  PROC DrawPart23()
    MoveL Offs(pOrigin,281.13,291.37,0.00),v40,z0,tPen\WObj:=wPaper;
    MoveL Offs(pOrigin,281.61,291.85,0.00),v40,z0,tPen\WObj:=wPaper;
    MoveL Offs(pOrigin,281.13,290.89,0.00),v40,z0,tPen\WObj:=wPaper;
    MoveL Offs(pOrigin,281.13,291.37,0.00),v40,z0,tPen\WObj:=wPaper;
    MoveL Offs(pOrigin,281.61,291.85,0.00),v40,fine,tPen\WObj:=wPaper;
    MoveL Offs(pOrigin,281.61,291.85,6.00),v60,z5,tPen\WObj:=wPaper;
    MoveL Offs(pOrigin,262.45,299.03,6.00),vTravel,z5,tPen\WObj:=wPaper;
    MoveL Offs(pOrigin,262.45,299.03,0.00),v60,z0,tPen\WObj:=wPaper;
    MoveL Offs(pOrigin,261.01,295.20,0.00),v40,z0,tPen\WObj:=wPaper;
    MoveL Offs(pOrigin,260.54,294.72,0.00),v40,z0,tPen\WObj:=wPaper;
    MoveL Offs(pOrigin,254.79,294.72,0.00),v40,z0,tPen\WObj:=wPaper;
    MoveL Offs(pOrigin,253.35,295.20,0.00),v40,z0,tPen\WObj:=wPaper;
    MoveL Offs(pOrigin,238.51,295.20,0.00),v40,z0,tPen\WObj:=wPaper;
    MoveL Offs(pOrigin,237.07,294.72,0.00),v40,z0,tPen\WObj:=wPaper;
    MoveL Offs(pOrigin,234.20,294.72,0.00),v40,z0,tPen\WObj:=wPaper;
    MoveL Offs(pOrigin,231.32,293.76,0.00),v40,z0,tPen\WObj:=wPaper;
    MoveL Offs(pOrigin,228.45,293.76,0.00),v40,z0,tPen\WObj:=wPaper;
    MoveL Offs(pOrigin,223.18,292.32,0.00),v40,z0,tPen\WObj:=wPaper;
    MoveL Offs(pOrigin,222.23,292.32,0.00),v40,z0,tPen\WObj:=wPaper;
    MoveL Offs(pOrigin,219.83,291.37,0.00),v40,z0,tPen\WObj:=wPaper;
    MoveL Offs(pOrigin,218.39,291.37,0.00),v40,z0,tPen\WObj:=wPaper;
    MoveL Offs(pOrigin,210.73,288.81,0.00),v40,z0,tPen\WObj:=wPaper;
    MoveL Offs(pOrigin,198.28,282.91,0.00),v40,z0,tPen\WObj:=wPaper;
    MoveL Offs(pOrigin,193.97,280.51,0.00),v40,z0,tPen\WObj:=wPaper;
    MoveL Offs(pOrigin,183.44,273.65,0.00),v40,z0,tPen\WObj:=wPaper;
    MoveL Offs(pOrigin,175.77,267.42,0.00),v40,z0,tPen\WObj:=wPaper;
    MoveL Offs(pOrigin,166.20,257.85,0.00),v40,z0,tPen\WObj:=wPaper;
    MoveL Offs(pOrigin,154.23,242.04,0.00),v40,z0,tPen\WObj:=wPaper;
    MoveL Offs(pOrigin,153.27,241.56,0.00),v40,z0,tPen\WObj:=wPaper;
    MoveL Offs(pOrigin,150.87,242.04,0.00),v40,z0,tPen\WObj:=wPaper;
    MoveL Offs(pOrigin,148.96,241.56,0.00),v40,z0,tPen\WObj:=wPaper;
    MoveL Offs(pOrigin,148.16,242.04,0.00),v40,z0,tPen\WObj:=wPaper;
    MoveL Offs(pOrigin,148.64,243.96,0.00),v40,z0,tPen\WObj:=wPaper;
    MoveL Offs(pOrigin,153.59,253.06,0.00),v40,z0,tPen\WObj:=wPaper;
    MoveL Offs(pOrigin,158.54,260.24,0.00),v40,z0,tPen\WObj:=wPaper;
    MoveL Offs(pOrigin,165.24,268.38,0.00),v40,z0,tPen\WObj:=wPaper;
    MoveL Offs(pOrigin,176.73,279.39,0.00),v40,z0,tPen\WObj:=wPaper;
    MoveL Offs(pOrigin,181.04,282.75,0.00),v40,z0,tPen\WObj:=wPaper;
    MoveL Offs(pOrigin,186.79,286.74,0.00),v40,z0,tPen\WObj:=wPaper;
    MoveL Offs(pOrigin,196.37,292.16,0.00),v40,z0,tPen\WObj:=wPaper;
    MoveL Offs(pOrigin,203.07,295.04,0.00),v40,z0,tPen\WObj:=wPaper;
    MoveL Offs(pOrigin,204.51,296.00,0.00),v40,z0,tPen\WObj:=wPaper;
    MoveL Offs(pOrigin,212.17,298.55,0.00),v40,z0,tPen\WObj:=wPaper;
    MoveL Offs(pOrigin,213.13,298.55,0.00),v40,z0,tPen\WObj:=wPaper;
    MoveL Offs(pOrigin,215.52,299.51,0.00),v40,z0,tPen\WObj:=wPaper;
    MoveL Offs(pOrigin,227.01,302.38,0.00),v40,z0,tPen\WObj:=wPaper;
    MoveL Offs(pOrigin,228.93,302.38,0.00),v40,z0,tPen\WObj:=wPaper;
    MoveL Offs(pOrigin,233.24,303.34,0.00),v40,z0,tPen\WObj:=wPaper;
    MoveL Offs(pOrigin,242.82,303.34,0.00),v40,z0,tPen\WObj:=wPaper;
    MoveL Offs(pOrigin,244.25,303.82,0.00),v40,z0,tPen\WObj:=wPaper;
    MoveL Offs(pOrigin,247.61,303.82,0.00),v40,z0,tPen\WObj:=wPaper;
    MoveL Offs(pOrigin,249.04,303.34,0.00),v40,z0,tPen\WObj:=wPaper;
    MoveL Offs(pOrigin,256.23,303.34,0.00),v40,z0,tPen\WObj:=wPaper;
    MoveL Offs(pOrigin,262.29,301.74,0.00),v40,z0,tPen\WObj:=wPaper;
    MoveL Offs(pOrigin,262.45,299.03,0.00),v40,fine,tPen\WObj:=wPaper;
    MoveL Offs(pOrigin,262.45,299.03,6.00),v60,z5,tPen\WObj:=wPaper;
    MoveL Offs(pOrigin,265.32,312.92,6.00),vTravel,z5,tPen\WObj:=wPaper;
    MoveL Offs(pOrigin,265.32,312.92,0.00),v60,z0,tPen\WObj:=wPaper;
    MoveL Offs(pOrigin,266.28,313.39,0.00),v40,z0,tPen\WObj:=wPaper;
    MoveL Offs(pOrigin,267.08,314.35,0.00),v40,z0,tPen\WObj:=wPaper;
    MoveL Offs(pOrigin,267.40,316.27,0.00),v40,z0,tPen\WObj:=wPaper;
    MoveL Offs(pOrigin,268.68,319.14,0.00),v40,z0,tPen\WObj:=wPaper;
    MoveL Offs(pOrigin,268.20,320.42,0.00),v40,z0,tPen\WObj:=wPaper;
    MoveL Offs(pOrigin,266.76,321.06,0.00),v40,z0,tPen\WObj:=wPaper;
    MoveL Offs(pOrigin,264.85,321.06,0.00),v40,z0,tPen\WObj:=wPaper;
    MoveL Offs(pOrigin,263.41,321.54,0.00),v40,z0,tPen\WObj:=wPaper;
    MoveL Offs(pOrigin,260.06,321.54,0.00),v40,z0,tPen\WObj:=wPaper;
    MoveL Offs(pOrigin,255.75,322.49,0.00),v40,z0,tPen\WObj:=wPaper;
    MoveL Offs(pOrigin,235.63,322.49,0.00),v40,z0,tPen\WObj:=wPaper;
    MoveL Offs(pOrigin,232.28,321.54,0.00),v40,z0,tPen\WObj:=wPaper;
    MoveL Offs(pOrigin,228.45,321.54,0.00),v40,z0,tPen\WObj:=wPaper;
    MoveL Offs(pOrigin,227.01,321.06,0.00),v40,z0,tPen\WObj:=wPaper;
    MoveL Offs(pOrigin,225.10,321.06,0.00),v40,z0,tPen\WObj:=wPaper;
    MoveL Offs(pOrigin,222.23,320.10,0.00),v40,z0,tPen\WObj:=wPaper;
    MoveL Offs(pOrigin,220.31,320.10,0.00),v40,z0,tPen\WObj:=wPaper;
    MoveL Offs(pOrigin,206.90,316.43,0.00),v40,z0,tPen\WObj:=wPaper;
    MoveL Offs(pOrigin,197.32,312.76,0.00),v40,z0,tPen\WObj:=wPaper;
    MoveL Offs(pOrigin,185.83,307.33,0.00),v40,z0,tPen\WObj:=wPaper;
    MoveL Offs(pOrigin,181.04,304.46,0.00),v40,z0,tPen\WObj:=wPaper;
    MoveL Offs(pOrigin,168.59,296.15,0.00),v40,z0,tPen\WObj:=wPaper;
    MoveL Offs(pOrigin,166.20,293.76,0.00),v40,z0,tPen\WObj:=wPaper;
    MoveL Offs(pOrigin,161.41,289.93,0.00),v40,z0,tPen\WObj:=wPaper;
    MoveL Offs(pOrigin,152.31,280.83,0.00),v40,z0,tPen\WObj:=wPaper;
    MoveL Offs(pOrigin,142.25,268.38,0.00),v40,z0,tPen\WObj:=wPaper;
    MoveL Offs(pOrigin,135.71,257.85,0.00),v40,z0,tPen\WObj:=wPaper;
    MoveL Offs(pOrigin,131.88,250.66,0.00),v40,z0,tPen\WObj:=wPaper;
    MoveL Offs(pOrigin,128.69,243.48,0.00),v40,z0,tPen\WObj:=wPaper;
    MoveL Offs(pOrigin,126.29,237.25,0.00),v40,z0,tPen\WObj:=wPaper;
    MoveL Offs(pOrigin,123.58,228.63,0.00),v40,z0,tPen\WObj:=wPaper;
    MoveL Offs(pOrigin,123.58,227.68,0.00),v40,z0,tPen\WObj:=wPaper;
    MoveL Offs(pOrigin,122.62,225.28,0.00),v40,z0,tPen\WObj:=wPaper;
    MoveL Offs(pOrigin,122.14,221.93,0.00),v40,z0,tPen\WObj:=wPaper;
    MoveL Offs(pOrigin,121.18,219.06,0.00),v40,z0,tPen\WObj:=wPaper;
    MoveL Offs(pOrigin,121.18,217.14,0.00),v40,z0,tPen\WObj:=wPaper;
    MoveL Offs(pOrigin,120.23,213.79,0.00),v40,z0,tPen\WObj:=wPaper;
    MoveL Offs(pOrigin,120.23,211.87,0.00),v40,z0,tPen\WObj:=wPaper;
    MoveL Offs(pOrigin,119.75,210.44,0.00),v40,z0,tPen\WObj:=wPaper;
    MoveL Offs(pOrigin,119.75,207.56,0.00),v40,z0,tPen\WObj:=wPaper;
    MoveL Offs(pOrigin,118.79,203.73,0.00),v40,z0,tPen\WObj:=wPaper;
    MoveL Offs(pOrigin,118.79,185.54,0.00),v40,z0,tPen\WObj:=wPaper;
    MoveL Offs(pOrigin,119.27,184.10,0.00),v40,z0,tPen\WObj:=wPaper;
    MoveL Offs(pOrigin,119.27,182.66,0.00),v40,z0,tPen\WObj:=wPaper;
    MoveL Offs(pOrigin,119.75,181.23,0.00),v40,z0,tPen\WObj:=wPaper;
    MoveL Offs(pOrigin,119.75,178.83,0.00),v40,z0,tPen\WObj:=wPaper;
    MoveL Offs(pOrigin,121.18,172.61,0.00),v40,z0,tPen\WObj:=wPaper;
    MoveL Offs(pOrigin,121.18,171.17,0.00),v40,z0,tPen\WObj:=wPaper;
    MoveL Offs(pOrigin,122.62,165.42,0.00),v40,z0,tPen\WObj:=wPaper;
    MoveL Offs(pOrigin,123.10,164.62,0.00),v40,z0,tPen\WObj:=wPaper;
    MoveL Offs(pOrigin,124.06,164.46,0.00),v40,z0,tPen\WObj:=wPaper;
    MoveL Offs(pOrigin,127.89,166.86,0.00),v40,z0,tPen\WObj:=wPaper;
    MoveL Offs(pOrigin,129.32,168.77,0.00),v40,z0,tPen\WObj:=wPaper;
    MoveL Offs(pOrigin,129.32,170.69,0.00),v40,z0,tPen\WObj:=wPaper;
    MoveL Offs(pOrigin,128.37,173.56,0.00),v40,z0,tPen\WObj:=wPaper;
    MoveL Offs(pOrigin,128.37,175.48,0.00),v40,z0,tPen\WObj:=wPaper;
    MoveL Offs(pOrigin,127.41,178.83,0.00),v40,z0,tPen\WObj:=wPaper;
    MoveL Offs(pOrigin,127.41,180.75,0.00),v40,z0,tPen\WObj:=wPaper;
    MoveL Offs(pOrigin,126.93,182.18,0.00),v40,z0,tPen\WObj:=wPaper;
    MoveL Offs(pOrigin,126.93,185.54,0.00),v40,z0,tPen\WObj:=wPaper;
    MoveL Offs(pOrigin,126.45,186.97,0.00),v40,z0,tPen\WObj:=wPaper;
    MoveL Offs(pOrigin,126.45,189.37,0.00),v40,z0,tPen\WObj:=wPaper;
  ENDPROC

  PROC DrawPart24()
    MoveL Offs(pOrigin,125.97,190.80,0.00),v40,z0,tPen\WObj:=wPaper;
    MoveL Offs(pOrigin,125.97,196.55,0.00),v40,z0,tPen\WObj:=wPaper;
    MoveL Offs(pOrigin,126.45,197.99,0.00),v40,z0,tPen\WObj:=wPaper;
    MoveL Offs(pOrigin,126.45,201.82,0.00),v40,z0,tPen\WObj:=wPaper;
    MoveL Offs(pOrigin,126.93,203.25,0.00),v40,z0,tPen\WObj:=wPaper;
    MoveL Offs(pOrigin,126.93,207.56,0.00),v40,z0,tPen\WObj:=wPaper;
    MoveL Offs(pOrigin,127.41,209.00,0.00),v40,z0,tPen\WObj:=wPaper;
    MoveL Offs(pOrigin,127.41,210.92,0.00),v40,z0,tPen\WObj:=wPaper;
    MoveL Offs(pOrigin,128.37,214.27,0.00),v40,z0,tPen\WObj:=wPaper;
    MoveL Offs(pOrigin,128.37,216.66,0.00),v40,z0,tPen\WObj:=wPaper;
    MoveL Offs(pOrigin,132.20,231.51,0.00),v40,z0,tPen\WObj:=wPaper;
    MoveL Offs(pOrigin,133.00,232.94,0.00),v40,z0,tPen\WObj:=wPaper;
    MoveL Offs(pOrigin,133.95,236.30,0.00),v40,z0,tPen\WObj:=wPaper;
    MoveL Offs(pOrigin,137.31,244.44,0.00),v40,z0,tPen\WObj:=wPaper;
    MoveL Offs(pOrigin,141.62,253.06,0.00),v40,z0,tPen\WObj:=wPaper;
    MoveL Offs(pOrigin,146.56,261.20,0.00),v40,z0,tPen\WObj:=wPaper;
    MoveL Offs(pOrigin,153.27,270.30,0.00),v40,z0,tPen\WObj:=wPaper;
    MoveL Offs(pOrigin,158.54,276.52,0.00),v40,z0,tPen\WObj:=wPaper;
    MoveL Offs(pOrigin,168.11,285.62,0.00),v40,z0,tPen\WObj:=wPaper;
    MoveL Offs(pOrigin,175.30,291.37,0.00),v40,z0,tPen\WObj:=wPaper;
    MoveL Offs(pOrigin,180.08,294.72,0.00),v40,z0,tPen\WObj:=wPaper;
    MoveL Offs(pOrigin,190.14,300.78,0.00),v40,z0,tPen\WObj:=wPaper;
    MoveL Offs(pOrigin,196.85,303.98,0.00),v40,z0,tPen\WObj:=wPaper;
    MoveL Offs(pOrigin,201.95,305.89,0.00),v40,z0,tPen\WObj:=wPaper;
    MoveL Offs(pOrigin,204.51,307.33,0.00),v40,z0,tPen\WObj:=wPaper;
    MoveL Offs(pOrigin,207.86,308.29,0.00),v40,z0,tPen\WObj:=wPaper;
    MoveL Offs(pOrigin,209.30,309.08,0.00),v40,z0,tPen\WObj:=wPaper;
    MoveL Offs(pOrigin,210.25,309.08,0.00),v40,z0,tPen\WObj:=wPaper;
    MoveL Offs(pOrigin,214.56,310.52,0.00),v40,z0,tPen\WObj:=wPaper;
    MoveL Offs(pOrigin,216.00,310.52,0.00),v40,z0,tPen\WObj:=wPaper;
    MoveL Offs(pOrigin,218.39,311.48,0.00),v40,z0,tPen\WObj:=wPaper;
    MoveL Offs(pOrigin,221.75,311.96,0.00),v40,z0,tPen\WObj:=wPaper;
    MoveL Offs(pOrigin,225.10,312.92,0.00),v40,z0,tPen\WObj:=wPaper;
    MoveL Offs(pOrigin,227.49,312.92,0.00),v40,z0,tPen\WObj:=wPaper;
    MoveL Offs(pOrigin,231.32,313.87,0.00),v40,z0,tPen\WObj:=wPaper;
    MoveL Offs(pOrigin,234.20,313.87,0.00),v40,z0,tPen\WObj:=wPaper;
    MoveL Offs(pOrigin,235.63,314.35,0.00),v40,z0,tPen\WObj:=wPaper;
    MoveL Offs(pOrigin,242.82,314.35,0.00),v40,z0,tPen\WObj:=wPaper;
    MoveL Offs(pOrigin,244.25,314.83,0.00),v40,z0,tPen\WObj:=wPaper;
    MoveL Offs(pOrigin,248.08,314.83,0.00),v40,z0,tPen\WObj:=wPaper;
    MoveL Offs(pOrigin,249.52,314.35,0.00),v40,z0,tPen\WObj:=wPaper;
    MoveL Offs(pOrigin,256.23,314.35,0.00),v40,z0,tPen\WObj:=wPaper;
    MoveL Offs(pOrigin,257.66,313.87,0.00),v40,z0,tPen\WObj:=wPaper;
    MoveL Offs(pOrigin,260.54,313.87,0.00),v40,z0,tPen\WObj:=wPaper;
    MoveL Offs(pOrigin,265.32,312.92,0.00),v40,fine,tPen\WObj:=wPaper;
    MoveL Offs(pOrigin,265.32,312.92,6.00),v60,z5,tPen\WObj:=wPaper;
    MoveL Offs(pOrigin,280.65,317.70,6.00),vTravel,z5,tPen\WObj:=wPaper;
    MoveL Offs(pOrigin,280.65,317.70,0.00),v60,z0,tPen\WObj:=wPaper;
    MoveL Offs(pOrigin,281.45,319.14,0.00),v40,z0,tPen\WObj:=wPaper;
    MoveL Offs(pOrigin,283.04,325.37,0.00),v40,z0,tPen\WObj:=wPaper;
    MoveL Offs(pOrigin,283.84,326.80,0.00),v40,z0,tPen\WObj:=wPaper;
    MoveL Offs(pOrigin,285.12,330.63,0.00),v40,z0,tPen\WObj:=wPaper;
    MoveL Offs(pOrigin,285.92,331.43,0.00),v40,z0,tPen\WObj:=wPaper;
    MoveL Offs(pOrigin,286.87,331.59,0.00),v40,z0,tPen\WObj:=wPaper;
    MoveL Offs(pOrigin,282.88,322.17,0.00),v40,z0,tPen\WObj:=wPaper;
    MoveL Offs(pOrigin,280.65,317.70,0.00),v40,fine,tPen\WObj:=wPaper;
    MoveL Offs(pOrigin,280.65,317.70,6.00),v60,z5,tPen\WObj:=wPaper;
    MoveL Offs(pOrigin,288.31,331.43,6.00),vTravel,z5,tPen\WObj:=wPaper;
    MoveL Offs(pOrigin,288.31,331.43,0.00),v60,z0,tPen\WObj:=wPaper;
    MoveL Offs(pOrigin,291.66,330.47,0.00),v40,z0,tPen\WObj:=wPaper;
    MoveL Offs(pOrigin,298.37,327.44,0.00),v40,z0,tPen\WObj:=wPaper;
    MoveL Offs(pOrigin,299.80,327.12,0.00),v40,z0,tPen\WObj:=wPaper;
    MoveL Offs(pOrigin,306.83,323.29,0.00),v40,z0,tPen\WObj:=wPaper;
    MoveL Offs(pOrigin,288.31,331.43,0.00),v40,fine,tPen\WObj:=wPaper;
    MoveL Offs(pOrigin,288.31,331.43,6.00),v60,z5,tPen\WObj:=wPaper;
    MoveL Offs(pOrigin,297.41,327.76,6.00),vTravel,z5,tPen\WObj:=wPaper;
    MoveL Offs(pOrigin,297.41,327.76,0.00),v60,z0,tPen\WObj:=wPaper;
    MoveL Offs(pOrigin,297.89,327.28,0.00),v40,z0,tPen\WObj:=wPaper;
    MoveL Offs(pOrigin,297.89,327.76,0.00),v40,z0,tPen\WObj:=wPaper;
    MoveL Offs(pOrigin,297.41,327.76,0.00),v40,z0,tPen\WObj:=wPaper;
    MoveL Offs(pOrigin,297.89,327.28,0.00),v40,z0,tPen\WObj:=wPaper;
    MoveL Offs(pOrigin,297.89,327.76,0.00),v40,z0,tPen\WObj:=wPaper;
    MoveL Offs(pOrigin,297.41,327.76,0.00),v40,fine,tPen\WObj:=wPaper;
    MoveL Offs(pOrigin,297.41,327.76,6.00),v60,z5,tPen\WObj:=wPaper;
    MoveL Offs(pOrigin,302.68,325.37,6.00),vTravel,z5,tPen\WObj:=wPaper;
    MoveL Offs(pOrigin,302.68,325.37,0.00),v60,z0,tPen\WObj:=wPaper;
    MoveL Offs(pOrigin,303.15,324.89,0.00),v40,z0,tPen\WObj:=wPaper;
    MoveL Offs(pOrigin,303.15,325.37,0.00),v40,z0,tPen\WObj:=wPaper;
    MoveL Offs(pOrigin,302.68,325.37,0.00),v40,z0,tPen\WObj:=wPaper;
    MoveL Offs(pOrigin,303.15,324.89,0.00),v40,z0,tPen\WObj:=wPaper;
    MoveL Offs(pOrigin,303.15,325.37,0.00),v40,z0,tPen\WObj:=wPaper;
    MoveL Offs(pOrigin,302.68,325.37,0.00),v40,fine,tPen\WObj:=wPaper;
    MoveL Offs(pOrigin,302.68,325.37,6.00),v60,z5,tPen\WObj:=wPaper;
    MoveL Offs(pOrigin,307.94,322.81,6.00),vTravel,z5,tPen\WObj:=wPaper;
    MoveL Offs(pOrigin,307.94,322.81,0.00),v60,z0,tPen\WObj:=wPaper;
    MoveL Offs(pOrigin,321.35,314.83,0.00),v40,z0,tPen\WObj:=wPaper;
    MoveL Offs(pOrigin,321.99,314.03,0.00),v40,z0,tPen\WObj:=wPaper;
    MoveL Offs(pOrigin,307.94,322.81,0.00),v40,fine,tPen\WObj:=wPaper;
    MoveL Offs(pOrigin,307.94,322.81,6.00),v60,z5,tPen\WObj:=wPaper;
    MoveL Offs(pOrigin,308.90,322.01,6.00),vTravel,z5,tPen\WObj:=wPaper;
    MoveL Offs(pOrigin,308.90,322.01,0.00),v60,z0,tPen\WObj:=wPaper;
    MoveL Offs(pOrigin,309.38,321.54,0.00),v40,z0,tPen\WObj:=wPaper;
    MoveL Offs(pOrigin,309.38,322.01,0.00),v40,z0,tPen\WObj:=wPaper;
    MoveL Offs(pOrigin,308.90,322.01,0.00),v40,z0,tPen\WObj:=wPaper;
    MoveL Offs(pOrigin,309.38,321.54,0.00),v40,z0,tPen\WObj:=wPaper;
    MoveL Offs(pOrigin,309.38,322.01,0.00),v40,z0,tPen\WObj:=wPaper;
    MoveL Offs(pOrigin,308.90,322.01,0.00),v40,fine,tPen\WObj:=wPaper;
    MoveL Offs(pOrigin,308.90,322.01,6.00),v60,z5,tPen\WObj:=wPaper;
    MoveL Offs(pOrigin,313.21,319.62,6.00),vTravel,z5,tPen\WObj:=wPaper;
    MoveL Offs(pOrigin,313.21,319.62,0.00),v60,z0,tPen\WObj:=wPaper;
    MoveL Offs(pOrigin,313.69,319.14,0.00),v40,z0,tPen\WObj:=wPaper;
    MoveL Offs(pOrigin,313.69,319.62,0.00),v40,z0,tPen\WObj:=wPaper;
    MoveL Offs(pOrigin,313.21,319.62,0.00),v40,z0,tPen\WObj:=wPaper;
    MoveL Offs(pOrigin,313.69,319.14,0.00),v40,z0,tPen\WObj:=wPaper;
    MoveL Offs(pOrigin,313.69,319.62,0.00),v40,z0,tPen\WObj:=wPaper;
    MoveL Offs(pOrigin,313.21,319.62,0.00),v40,fine,tPen\WObj:=wPaper;
    MoveL Offs(pOrigin,313.21,319.62,6.00),v60,z5,tPen\WObj:=wPaper;
    MoveL Offs(pOrigin,314.65,318.66,6.00),vTravel,z5,tPen\WObj:=wPaper;
    MoveL Offs(pOrigin,314.65,318.66,0.00),v60,z0,tPen\WObj:=wPaper;
    MoveL Offs(pOrigin,315.13,318.18,0.00),v40,z0,tPen\WObj:=wPaper;
    MoveL Offs(pOrigin,315.13,318.66,0.00),v40,z0,tPen\WObj:=wPaper;
    MoveL Offs(pOrigin,314.65,318.66,0.00),v40,z0,tPen\WObj:=wPaper;
    MoveL Offs(pOrigin,315.13,318.18,0.00),v40,z0,tPen\WObj:=wPaper;
    MoveL Offs(pOrigin,315.13,318.66,0.00),v40,z0,tPen\WObj:=wPaper;
    MoveL Offs(pOrigin,314.65,318.66,0.00),v40,fine,tPen\WObj:=wPaper;
    MoveL Offs(pOrigin,314.65,318.66,6.00),v60,z5,tPen\WObj:=wPaper;
    MoveL Offs(pOrigin,317.04,317.23,6.00),vTravel,z5,tPen\WObj:=wPaper;
    MoveL Offs(pOrigin,317.04,317.23,0.00),v60,z0,tPen\WObj:=wPaper;
    MoveL Offs(pOrigin,317.52,316.75,0.00),v40,z0,tPen\WObj:=wPaper;
    MoveL Offs(pOrigin,317.52,317.23,0.00),v40,z0,tPen\WObj:=wPaper;
  ENDPROC

  PROC DrawPart25()
    MoveL Offs(pOrigin,317.04,317.23,0.00),v40,z0,tPen\WObj:=wPaper;
    MoveL Offs(pOrigin,317.52,316.75,0.00),v40,z0,tPen\WObj:=wPaper;
    MoveL Offs(pOrigin,317.52,317.23,0.00),v40,z0,tPen\WObj:=wPaper;
    MoveL Offs(pOrigin,317.04,317.23,0.00),v40,fine,tPen\WObj:=wPaper;
    MoveL Offs(pOrigin,317.04,317.23,6.00),v60,z5,tPen\WObj:=wPaper;
    MoveL Offs(pOrigin,312.25,310.04,6.00),vTravel,z5,tPen\WObj:=wPaper;
    MoveL Offs(pOrigin,312.25,310.04,0.00),v60,z0,tPen\WObj:=wPaper;
    MoveL Offs(pOrigin,311.77,310.04,0.00),v40,z0,tPen\WObj:=wPaper;
    MoveL Offs(pOrigin,312.25,309.56,0.00),v40,z0,tPen\WObj:=wPaper;
    MoveL Offs(pOrigin,312.25,310.04,0.00),v40,z0,tPen\WObj:=wPaper;
    MoveL Offs(pOrigin,311.77,310.04,0.00),v40,z0,tPen\WObj:=wPaper;
    MoveL Offs(pOrigin,312.25,309.56,0.00),v40,z0,tPen\WObj:=wPaper;
    MoveL Offs(pOrigin,312.25,310.04,0.00),v40,fine,tPen\WObj:=wPaper;
    MoveL Offs(pOrigin,312.25,310.04,6.00),v60,z5,tPen\WObj:=wPaper;
    MoveL Offs(pOrigin,310.82,310.52,6.00),vTravel,z5,tPen\WObj:=wPaper;
    MoveL Offs(pOrigin,310.82,310.52,0.00),v60,z0,tPen\WObj:=wPaper;
    MoveL Offs(pOrigin,310.82,311.00,0.00),v40,z0,tPen\WObj:=wPaper;
    MoveL Offs(pOrigin,310.34,311.00,0.00),v40,z0,tPen\WObj:=wPaper;
    MoveL Offs(pOrigin,310.82,310.52,0.00),v40,z0,tPen\WObj:=wPaper;
    MoveL Offs(pOrigin,310.82,311.00,0.00),v40,z0,tPen\WObj:=wPaper;
    MoveL Offs(pOrigin,310.34,311.00,0.00),v40,z0,tPen\WObj:=wPaper;
    MoveL Offs(pOrigin,310.82,310.52,0.00),v40,fine,tPen\WObj:=wPaper;
    MoveL Offs(pOrigin,310.82,310.52,6.00),v60,z5,tPen\WObj:=wPaper;
    MoveL Offs(pOrigin,317.04,306.69,6.00),vTravel,z5,tPen\WObj:=wPaper;
    MoveL Offs(pOrigin,317.04,306.69,0.00),v60,z0,tPen\WObj:=wPaper;
    MoveL Offs(pOrigin,318.00,305.73,0.00),v40,z0,tPen\WObj:=wPaper;
    MoveL Offs(pOrigin,318.00,306.21,0.00),v40,z0,tPen\WObj:=wPaper;
    MoveL Offs(pOrigin,317.52,306.21,0.00),v40,z0,tPen\WObj:=wPaper;
    MoveL Offs(pOrigin,317.04,306.69,0.00),v40,z0,tPen\WObj:=wPaper;
    MoveL Offs(pOrigin,318.00,305.73,0.00),v40,z0,tPen\WObj:=wPaper;
    MoveL Offs(pOrigin,318.00,306.21,0.00),v40,z0,tPen\WObj:=wPaper;
    MoveL Offs(pOrigin,317.52,306.21,0.00),v40,z0,tPen\WObj:=wPaper;
    MoveL Offs(pOrigin,317.04,306.69,0.00),v40,fine,tPen\WObj:=wPaper;
    MoveL Offs(pOrigin,317.04,306.69,6.00),v60,z5,tPen\WObj:=wPaper;
    MoveL Offs(pOrigin,318.96,305.25,6.00),vTravel,z5,tPen\WObj:=wPaper;
    MoveL Offs(pOrigin,318.96,305.25,0.00),v60,z0,tPen\WObj:=wPaper;
    MoveL Offs(pOrigin,319.44,304.77,0.00),v40,z0,tPen\WObj:=wPaper;
    MoveL Offs(pOrigin,319.44,305.25,0.00),v40,z0,tPen\WObj:=wPaper;
    MoveL Offs(pOrigin,318.96,305.25,0.00),v40,z0,tPen\WObj:=wPaper;
    MoveL Offs(pOrigin,319.44,304.77,0.00),v40,z0,tPen\WObj:=wPaper;
    MoveL Offs(pOrigin,319.44,305.25,0.00),v40,z0,tPen\WObj:=wPaper;
    MoveL Offs(pOrigin,318.96,305.25,0.00),v40,fine,tPen\WObj:=wPaper;
    MoveL Offs(pOrigin,318.96,305.25,6.00),v60,z5,tPen\WObj:=wPaper;
    MoveL Offs(pOrigin,320.39,304.30,6.00),vTravel,z5,tPen\WObj:=wPaper;
    MoveL Offs(pOrigin,320.39,304.30,0.00),v60,z0,tPen\WObj:=wPaper;
    MoveL Offs(pOrigin,321.35,303.34,0.00),v40,z0,tPen\WObj:=wPaper;
    MoveL Offs(pOrigin,321.35,303.82,0.00),v40,z0,tPen\WObj:=wPaper;
    MoveL Offs(pOrigin,320.87,303.82,0.00),v40,z0,tPen\WObj:=wPaper;
    MoveL Offs(pOrigin,320.39,304.30,0.00),v40,z0,tPen\WObj:=wPaper;
    MoveL Offs(pOrigin,321.35,303.34,0.00),v40,z0,tPen\WObj:=wPaper;
    MoveL Offs(pOrigin,321.35,303.82,0.00),v40,z0,tPen\WObj:=wPaper;
    MoveL Offs(pOrigin,320.87,303.82,0.00),v40,z0,tPen\WObj:=wPaper;
    MoveL Offs(pOrigin,320.39,304.30,0.00),v40,fine,tPen\WObj:=wPaper;
    MoveL Offs(pOrigin,320.39,304.30,6.00),v60,z5,tPen\WObj:=wPaper;
    MoveL Offs(pOrigin,322.79,302.38,6.00),vTravel,z5,tPen\WObj:=wPaper;
    MoveL Offs(pOrigin,322.79,302.38,0.00),v60,z0,tPen\WObj:=wPaper;
    MoveL Offs(pOrigin,323.75,301.42,0.00),v40,z0,tPen\WObj:=wPaper;
    MoveL Offs(pOrigin,323.75,301.90,0.00),v40,z0,tPen\WObj:=wPaper;
    MoveL Offs(pOrigin,323.27,301.90,0.00),v40,z0,tPen\WObj:=wPaper;
    MoveL Offs(pOrigin,322.79,302.38,0.00),v40,z0,tPen\WObj:=wPaper;
    MoveL Offs(pOrigin,323.75,301.42,0.00),v40,z0,tPen\WObj:=wPaper;
    MoveL Offs(pOrigin,323.75,301.90,0.00),v40,z0,tPen\WObj:=wPaper;
    MoveL Offs(pOrigin,323.27,301.90,0.00),v40,z0,tPen\WObj:=wPaper;
    MoveL Offs(pOrigin,322.79,302.38,0.00),v40,fine,tPen\WObj:=wPaper;
    MoveL Offs(pOrigin,322.79,302.38,6.00),v60,z5,tPen\WObj:=wPaper;
    MoveL Offs(pOrigin,324.70,300.94,6.00),vTravel,z5,tPen\WObj:=wPaper;
    MoveL Offs(pOrigin,324.70,300.94,0.00),v60,z0,tPen\WObj:=wPaper;
    MoveL Offs(pOrigin,325.66,299.99,0.00),v40,z0,tPen\WObj:=wPaper;
    MoveL Offs(pOrigin,325.66,300.46,0.00),v40,z0,tPen\WObj:=wPaper;
    MoveL Offs(pOrigin,325.18,300.46,0.00),v40,z0,tPen\WObj:=wPaper;
    MoveL Offs(pOrigin,324.70,300.94,0.00),v40,z0,tPen\WObj:=wPaper;
    MoveL Offs(pOrigin,325.66,299.99,0.00),v40,z0,tPen\WObj:=wPaper;
    MoveL Offs(pOrigin,325.66,300.46,0.00),v40,z0,tPen\WObj:=wPaper;
    MoveL Offs(pOrigin,325.18,300.46,0.00),v40,z0,tPen\WObj:=wPaper;
    MoveL Offs(pOrigin,324.70,300.94,0.00),v40,fine,tPen\WObj:=wPaper;
    MoveL Offs(pOrigin,324.70,300.94,6.00),v60,z5,tPen\WObj:=wPaper;
    MoveL Offs(pOrigin,331.89,306.21,6.00),vTravel,z5,tPen\WObj:=wPaper;
    MoveL Offs(pOrigin,331.89,306.21,0.00),v60,z0,tPen\WObj:=wPaper;
    MoveL Offs(pOrigin,331.89,306.69,0.00),v40,z0,tPen\WObj:=wPaper;
    MoveL Offs(pOrigin,331.41,307.17,0.00),v40,z0,tPen\WObj:=wPaper;
    MoveL Offs(pOrigin,331.89,306.21,0.00),v40,z0,tPen\WObj:=wPaper;
    MoveL Offs(pOrigin,331.89,306.69,0.00),v40,z0,tPen\WObj:=wPaper;
    MoveL Offs(pOrigin,331.41,307.17,0.00),v40,z0,tPen\WObj:=wPaper;
    MoveL Offs(pOrigin,331.89,306.21,0.00),v40,z0,tPen\WObj:=wPaper;
    MoveL Offs(pOrigin,332.85,305.73,0.00),v40,z0,tPen\WObj:=wPaper;
    MoveL Offs(pOrigin,333.80,304.77,0.00),v40,z0,tPen\WObj:=wPaper;
    MoveL Offs(pOrigin,332.85,305.73,0.00),v40,fine,tPen\WObj:=wPaper;
    MoveL Offs(pOrigin,332.85,305.73,6.00),v60,z5,tPen\WObj:=wPaper;
    MoveL Offs(pOrigin,334.76,304.30,6.00),vTravel,z5,tPen\WObj:=wPaper;
    MoveL Offs(pOrigin,334.76,304.30,0.00),v60,z0,tPen\WObj:=wPaper;
    MoveL Offs(pOrigin,335.24,303.82,0.00),v40,z0,tPen\WObj:=wPaper;
    MoveL Offs(pOrigin,335.24,303.34,0.00),v40,z0,tPen\WObj:=wPaper;
    MoveL Offs(pOrigin,334.76,304.30,0.00),v40,z0,tPen\WObj:=wPaper;
    MoveL Offs(pOrigin,335.24,303.82,0.00),v40,z0,tPen\WObj:=wPaper;
    MoveL Offs(pOrigin,335.24,303.34,0.00),v40,z0,tPen\WObj:=wPaper;
    MoveL Offs(pOrigin,334.76,304.30,0.00),v40,fine,tPen\WObj:=wPaper;
    MoveL Offs(pOrigin,334.76,304.30,6.00),v60,z5,tPen\WObj:=wPaper;
    MoveL Offs(pOrigin,336.20,302.86,6.00),vTravel,z5,tPen\WObj:=wPaper;
    MoveL Offs(pOrigin,336.20,302.86,0.00),v60,z0,tPen\WObj:=wPaper;
    MoveL Offs(pOrigin,336.68,302.38,0.00),v40,z0,tPen\WObj:=wPaper;
    MoveL Offs(pOrigin,336.68,301.90,0.00),v40,z0,tPen\WObj:=wPaper;
    MoveL Offs(pOrigin,336.20,302.86,0.00),v40,z0,tPen\WObj:=wPaper;
    MoveL Offs(pOrigin,336.68,302.38,0.00),v40,z0,tPen\WObj:=wPaper;
    MoveL Offs(pOrigin,336.68,301.90,0.00),v40,z0,tPen\WObj:=wPaper;
    MoveL Offs(pOrigin,336.20,302.86,0.00),v40,fine,tPen\WObj:=wPaper;
    MoveL Offs(pOrigin,336.20,302.86,6.00),v60,z5,tPen\WObj:=wPaper;
    MoveL Offs(pOrigin,338.59,300.94,6.00),vTravel,z5,tPen\WObj:=wPaper;
    MoveL Offs(pOrigin,338.59,300.94,0.00),v60,z0,tPen\WObj:=wPaper;
    MoveL Offs(pOrigin,339.07,300.46,0.00),v40,z0,tPen\WObj:=wPaper;
    MoveL Offs(pOrigin,339.07,299.99,0.00),v40,z0,tPen\WObj:=wPaper;
    MoveL Offs(pOrigin,338.59,300.94,0.00),v40,z0,tPen\WObj:=wPaper;
    MoveL Offs(pOrigin,339.07,300.46,0.00),v40,z0,tPen\WObj:=wPaper;
    MoveL Offs(pOrigin,339.07,299.99,0.00),v40,z0,tPen\WObj:=wPaper;
    MoveL Offs(pOrigin,338.59,300.94,0.00),v40,fine,tPen\WObj:=wPaper;
    MoveL Offs(pOrigin,338.59,300.94,6.00),v60,z5,tPen\WObj:=wPaper;
    MoveL Offs(pOrigin,340.03,299.51,6.00),vTravel,z5,tPen\WObj:=wPaper;
    MoveL Offs(pOrigin,340.03,299.51,0.00),v60,z0,tPen\WObj:=wPaper;
    MoveL Offs(pOrigin,340.51,299.03,0.00),v40,z0,tPen\WObj:=wPaper;
    MoveL Offs(pOrigin,340.51,298.55,0.00),v40,z0,tPen\WObj:=wPaper;
    MoveL Offs(pOrigin,340.03,299.51,0.00),v40,z0,tPen\WObj:=wPaper;
  ENDPROC

  PROC DrawPart26()
    MoveL Offs(pOrigin,340.51,299.03,0.00),v40,z0,tPen\WObj:=wPaper;
    MoveL Offs(pOrigin,340.51,298.55,0.00),v40,z0,tPen\WObj:=wPaper;
    MoveL Offs(pOrigin,340.03,299.51,0.00),v40,fine,tPen\WObj:=wPaper;
    MoveL Offs(pOrigin,340.03,299.51,6.00),v60,z5,tPen\WObj:=wPaper;
    MoveL Offs(pOrigin,341.46,298.07,6.00),vTravel,z5,tPen\WObj:=wPaper;
    MoveL Offs(pOrigin,341.46,298.07,0.00),v60,z0,tPen\WObj:=wPaper;
    MoveL Offs(pOrigin,341.94,297.59,0.00),v40,z0,tPen\WObj:=wPaper;
    MoveL Offs(pOrigin,341.94,297.11,0.00),v40,z0,tPen\WObj:=wPaper;
    MoveL Offs(pOrigin,341.46,298.07,0.00),v40,z0,tPen\WObj:=wPaper;
    MoveL Offs(pOrigin,341.94,297.59,0.00),v40,z0,tPen\WObj:=wPaper;
    MoveL Offs(pOrigin,341.94,297.11,0.00),v40,z0,tPen\WObj:=wPaper;
    MoveL Offs(pOrigin,341.46,298.07,0.00),v40,fine,tPen\WObj:=wPaper;
    MoveL Offs(pOrigin,341.46,298.07,6.00),v60,z5,tPen\WObj:=wPaper;
    MoveL Offs(pOrigin,342.90,296.63,6.00),vTravel,z5,tPen\WObj:=wPaper;
    MoveL Offs(pOrigin,342.90,296.63,0.00),v60,z0,tPen\WObj:=wPaper;
    MoveL Offs(pOrigin,343.38,296.15,0.00),v40,z0,tPen\WObj:=wPaper;
    MoveL Offs(pOrigin,343.38,295.68,0.00),v40,z0,tPen\WObj:=wPaper;
    MoveL Offs(pOrigin,342.90,296.63,0.00),v40,z0,tPen\WObj:=wPaper;
    MoveL Offs(pOrigin,343.38,296.15,0.00),v40,z0,tPen\WObj:=wPaper;
    MoveL Offs(pOrigin,343.38,295.68,0.00),v40,z0,tPen\WObj:=wPaper;
    MoveL Offs(pOrigin,342.90,296.63,0.00),v40,fine,tPen\WObj:=wPaper;
    MoveL Offs(pOrigin,342.90,296.63,6.00),v60,z5,tPen\WObj:=wPaper;
    MoveL Offs(pOrigin,345.30,293.76,6.00),vTravel,z5,tPen\WObj:=wPaper;
    MoveL Offs(pOrigin,345.30,293.76,0.00),v60,z0,tPen\WObj:=wPaper;
    MoveL Offs(pOrigin,345.77,292.80,0.00),v40,z0,tPen\WObj:=wPaper;
    MoveL Offs(pOrigin,345.77,293.28,0.00),v40,z0,tPen\WObj:=wPaper;
    MoveL Offs(pOrigin,345.30,293.76,0.00),v40,z0,tPen\WObj:=wPaper;
    MoveL Offs(pOrigin,345.77,292.80,0.00),v40,z0,tPen\WObj:=wPaper;
    MoveL Offs(pOrigin,345.77,293.28,0.00),v40,z0,tPen\WObj:=wPaper;
    MoveL Offs(pOrigin,345.30,293.76,0.00),v40,fine,tPen\WObj:=wPaper;
    MoveL Offs(pOrigin,345.30,293.76,6.00),v60,z5,tPen\WObj:=wPaper;
    MoveL Offs(pOrigin,347.69,290.89,6.00),vTravel,z5,tPen\WObj:=wPaper;
    MoveL Offs(pOrigin,347.69,290.89,0.00),v60,z0,tPen\WObj:=wPaper;
    MoveL Offs(pOrigin,348.17,290.41,0.00),v40,z0,tPen\WObj:=wPaper;
    MoveL Offs(pOrigin,348.17,289.93,0.00),v40,z0,tPen\WObj:=wPaper;
    MoveL Offs(pOrigin,347.69,290.89,0.00),v40,z0,tPen\WObj:=wPaper;
    MoveL Offs(pOrigin,348.17,290.41,0.00),v40,z0,tPen\WObj:=wPaper;
    MoveL Offs(pOrigin,348.17,289.93,0.00),v40,z0,tPen\WObj:=wPaper;
    MoveL Offs(pOrigin,347.69,290.89,0.00),v40,fine,tPen\WObj:=wPaper;
    MoveL Offs(pOrigin,347.69,290.89,6.00),v60,z5,tPen\WObj:=wPaper;
    MoveL Offs(pOrigin,349.13,289.45,6.00),vTravel,z5,tPen\WObj:=wPaper;
    MoveL Offs(pOrigin,349.13,289.45,0.00),v60,z0,tPen\WObj:=wPaper;
    MoveL Offs(pOrigin,349.61,288.49,0.00),v40,z0,tPen\WObj:=wPaper;
    MoveL Offs(pOrigin,349.61,288.97,0.00),v40,z0,tPen\WObj:=wPaper;
    MoveL Offs(pOrigin,349.13,289.45,0.00),v40,z0,tPen\WObj:=wPaper;
    MoveL Offs(pOrigin,349.61,288.49,0.00),v40,z0,tPen\WObj:=wPaper;
    MoveL Offs(pOrigin,349.61,288.97,0.00),v40,z0,tPen\WObj:=wPaper;
    MoveL Offs(pOrigin,349.13,289.45,0.00),v40,fine,tPen\WObj:=wPaper;
    MoveL Offs(pOrigin,349.13,289.45,6.00),v60,z5,tPen\WObj:=wPaper;
    MoveL Offs(pOrigin,350.56,287.54,6.00),vTravel,z5,tPen\WObj:=wPaper;
    MoveL Offs(pOrigin,350.56,287.54,0.00),v60,z0,tPen\WObj:=wPaper;
    MoveL Offs(pOrigin,351.04,286.58,0.00),v40,z0,tPen\WObj:=wPaper;
    MoveL Offs(pOrigin,351.04,287.06,0.00),v40,z0,tPen\WObj:=wPaper;
    MoveL Offs(pOrigin,350.56,287.54,0.00),v40,z0,tPen\WObj:=wPaper;
    MoveL Offs(pOrigin,351.04,286.58,0.00),v40,z0,tPen\WObj:=wPaper;
    MoveL Offs(pOrigin,351.04,287.06,0.00),v40,z0,tPen\WObj:=wPaper;
    MoveL Offs(pOrigin,350.56,287.54,0.00),v40,fine,tPen\WObj:=wPaper;
    MoveL Offs(pOrigin,350.56,287.54,6.00),v60,z5,tPen\WObj:=wPaper;
    MoveL Offs(pOrigin,352.00,285.14,6.00),vTravel,z5,tPen\WObj:=wPaper;
    MoveL Offs(pOrigin,352.00,285.14,0.00),v60,z0,tPen\WObj:=wPaper;
    MoveL Offs(pOrigin,352.48,284.18,0.00),v40,z0,tPen\WObj:=wPaper;
    MoveL Offs(pOrigin,352.48,284.66,0.00),v40,z0,tPen\WObj:=wPaper;
    MoveL Offs(pOrigin,352.00,285.14,0.00),v40,z0,tPen\WObj:=wPaper;
    MoveL Offs(pOrigin,352.48,284.18,0.00),v40,z0,tPen\WObj:=wPaper;
    MoveL Offs(pOrigin,352.48,284.66,0.00),v40,z0,tPen\WObj:=wPaper;
    MoveL Offs(pOrigin,352.00,285.14,0.00),v40,fine,tPen\WObj:=wPaper;
    MoveL Offs(pOrigin,352.00,285.14,6.00),v60,z5,tPen\WObj:=wPaper;
    MoveL Offs(pOrigin,353.44,283.70,6.00),vTravel,z5,tPen\WObj:=wPaper;
    MoveL Offs(pOrigin,353.44,283.70,0.00),v60,z0,tPen\WObj:=wPaper;
    MoveL Offs(pOrigin,353.92,282.75,0.00),v40,z0,tPen\WObj:=wPaper;
    MoveL Offs(pOrigin,353.92,283.23,0.00),v40,z0,tPen\WObj:=wPaper;
    MoveL Offs(pOrigin,353.44,283.70,0.00),v40,z0,tPen\WObj:=wPaper;
    MoveL Offs(pOrigin,353.92,282.75,0.00),v40,z0,tPen\WObj:=wPaper;
    MoveL Offs(pOrigin,353.92,283.23,0.00),v40,z0,tPen\WObj:=wPaper;
    MoveL Offs(pOrigin,353.44,283.70,0.00),v40,fine,tPen\WObj:=wPaper;
    MoveL Offs(pOrigin,353.44,283.70,6.00),v60,z5,tPen\WObj:=wPaper;
    MoveL Offs(pOrigin,355.83,280.35,6.00),vTravel,z5,tPen\WObj:=wPaper;
    MoveL Offs(pOrigin,355.83,280.35,0.00),v60,z0,tPen\WObj:=wPaper;
    MoveL Offs(pOrigin,356.31,279.87,0.00),v40,z0,tPen\WObj:=wPaper;
    MoveL Offs(pOrigin,356.31,279.39,0.00),v40,z0,tPen\WObj:=wPaper;
    MoveL Offs(pOrigin,355.83,280.35,0.00),v40,z0,tPen\WObj:=wPaper;
    MoveL Offs(pOrigin,356.31,279.87,0.00),v40,z0,tPen\WObj:=wPaper;
    MoveL Offs(pOrigin,356.31,279.39,0.00),v40,z0,tPen\WObj:=wPaper;
    MoveL Offs(pOrigin,355.83,280.35,0.00),v40,fine,tPen\WObj:=wPaper;
    MoveL Offs(pOrigin,355.83,280.35,6.00),v60,z5,tPen\WObj:=wPaper;
    MoveL Offs(pOrigin,360.14,273.17,6.00),vTravel,z5,tPen\WObj:=wPaper;
    MoveL Offs(pOrigin,360.14,273.17,0.00),v60,z0,tPen\WObj:=wPaper;
    MoveL Offs(pOrigin,360.62,272.21,0.00),v40,z0,tPen\WObj:=wPaper;
    MoveL Offs(pOrigin,360.62,272.69,0.00),v40,z0,tPen\WObj:=wPaper;
    MoveL Offs(pOrigin,360.14,273.17,0.00),v40,z0,tPen\WObj:=wPaper;
    MoveL Offs(pOrigin,360.62,272.21,0.00),v40,z0,tPen\WObj:=wPaper;
    MoveL Offs(pOrigin,360.62,272.69,0.00),v40,z0,tPen\WObj:=wPaper;
    MoveL Offs(pOrigin,360.14,273.17,0.00),v40,fine,tPen\WObj:=wPaper;
    MoveL Offs(pOrigin,360.14,273.17,6.00),v60,z5,tPen\WObj:=wPaper;
    MoveL Offs(pOrigin,349.61,273.17,6.00),vTravel,z5,tPen\WObj:=wPaper;
    MoveL Offs(pOrigin,349.61,273.17,0.00),v60,z0,tPen\WObj:=wPaper;
    MoveL Offs(pOrigin,348.65,274.13,0.00),v40,z0,tPen\WObj:=wPaper;
    MoveL Offs(pOrigin,349.61,272.69,0.00),v40,z0,tPen\WObj:=wPaper;
    MoveL Offs(pOrigin,349.61,273.17,0.00),v40,z0,tPen\WObj:=wPaper;
    MoveL Offs(pOrigin,348.65,274.13,0.00),v40,z0,tPen\WObj:=wPaper;
    MoveL Offs(pOrigin,349.61,272.69,0.00),v40,z0,tPen\WObj:=wPaper;
    MoveL Offs(pOrigin,349.61,273.17,0.00),v40,fine,tPen\WObj:=wPaper;
    MoveL Offs(pOrigin,349.61,273.17,6.00),v60,z5,tPen\WObj:=wPaper;
    MoveL Offs(pOrigin,348.17,275.08,6.00),vTravel,z5,tPen\WObj:=wPaper;
    MoveL Offs(pOrigin,348.17,275.08,0.00),v60,z0,tPen\WObj:=wPaper;
    MoveL Offs(pOrigin,348.17,275.56,0.00),v40,z0,tPen\WObj:=wPaper;
    MoveL Offs(pOrigin,347.69,276.04,0.00),v40,z0,tPen\WObj:=wPaper;
    MoveL Offs(pOrigin,348.17,275.08,0.00),v40,z0,tPen\WObj:=wPaper;
    MoveL Offs(pOrigin,348.17,275.56,0.00),v40,z0,tPen\WObj:=wPaper;
    MoveL Offs(pOrigin,347.69,276.04,0.00),v40,z0,tPen\WObj:=wPaper;
    MoveL Offs(pOrigin,348.17,275.08,0.00),v40,fine,tPen\WObj:=wPaper;
    MoveL Offs(pOrigin,348.17,275.08,6.00),v60,z5,tPen\WObj:=wPaper;
    MoveL Offs(pOrigin,347.21,276.52,6.00),vTravel,z5,tPen\WObj:=wPaper;
    MoveL Offs(pOrigin,347.21,276.52,0.00),v60,z0,tPen\WObj:=wPaper;
    MoveL Offs(pOrigin,347.21,277.00,0.00),v40,z0,tPen\WObj:=wPaper;
    MoveL Offs(pOrigin,346.25,277.96,0.00),v40,z0,tPen\WObj:=wPaper;
    MoveL Offs(pOrigin,347.21,276.52,0.00),v40,z0,tPen\WObj:=wPaper;
    MoveL Offs(pOrigin,347.21,277.00,0.00),v40,z0,tPen\WObj:=wPaper;
    MoveL Offs(pOrigin,346.25,277.96,0.00),v40,z0,tPen\WObj:=wPaper;
    MoveL Offs(pOrigin,347.21,276.52,0.00),v40,fine,tPen\WObj:=wPaper;
  ENDPROC

  PROC DrawPart27()
    MoveL Offs(pOrigin,347.21,276.52,6.00),v60,z5,tPen\WObj:=wPaper;
    MoveL Offs(pOrigin,344.34,280.83,6.00),vTravel,z5,tPen\WObj:=wPaper;
    MoveL Offs(pOrigin,344.34,280.83,0.00),v60,z0,tPen\WObj:=wPaper;
    MoveL Offs(pOrigin,344.34,281.31,0.00),v40,z0,tPen\WObj:=wPaper;
    MoveL Offs(pOrigin,343.86,281.31,0.00),v40,z0,tPen\WObj:=wPaper;
    MoveL Offs(pOrigin,342.90,282.27,0.00),v40,z0,tPen\WObj:=wPaper;
    MoveL Offs(pOrigin,344.34,280.83,0.00),v40,z0,tPen\WObj:=wPaper;
    MoveL Offs(pOrigin,344.34,281.31,0.00),v40,z0,tPen\WObj:=wPaper;
    MoveL Offs(pOrigin,343.86,281.31,0.00),v40,z0,tPen\WObj:=wPaper;
    MoveL Offs(pOrigin,342.90,282.27,0.00),v40,z0,tPen\WObj:=wPaper;
    MoveL Offs(pOrigin,344.34,280.83,0.00),v40,fine,tPen\WObj:=wPaper;
    MoveL Offs(pOrigin,344.34,280.83,6.00),v60,z5,tPen\WObj:=wPaper;
    MoveL Offs(pOrigin,341.46,284.18,6.00),vTravel,z5,tPen\WObj:=wPaper;
    MoveL Offs(pOrigin,341.46,284.18,0.00),v60,z0,tPen\WObj:=wPaper;
    MoveL Offs(pOrigin,341.46,284.66,0.00),v40,z0,tPen\WObj:=wPaper;
    MoveL Offs(pOrigin,340.99,284.66,0.00),v40,z0,tPen\WObj:=wPaper;
    MoveL Offs(pOrigin,341.46,284.18,0.00),v40,z0,tPen\WObj:=wPaper;
    MoveL Offs(pOrigin,341.46,284.66,0.00),v40,z0,tPen\WObj:=wPaper;
    MoveL Offs(pOrigin,340.99,284.66,0.00),v40,z0,tPen\WObj:=wPaper;
    MoveL Offs(pOrigin,341.46,284.18,0.00),v40,fine,tPen\WObj:=wPaper;
    MoveL Offs(pOrigin,341.46,284.18,6.00),v60,z5,tPen\WObj:=wPaper;
    MoveL Offs(pOrigin,340.51,285.14,6.00),vTravel,z5,tPen\WObj:=wPaper;
    MoveL Offs(pOrigin,340.51,285.14,0.00),v60,z0,tPen\WObj:=wPaper;
    MoveL Offs(pOrigin,340.51,285.62,0.00),v40,z0,tPen\WObj:=wPaper;
    MoveL Offs(pOrigin,340.03,285.62,0.00),v40,z0,tPen\WObj:=wPaper;
    MoveL Offs(pOrigin,340.51,285.14,0.00),v40,z0,tPen\WObj:=wPaper;
    MoveL Offs(pOrigin,340.51,285.62,0.00),v40,z0,tPen\WObj:=wPaper;
    MoveL Offs(pOrigin,340.03,285.62,0.00),v40,z0,tPen\WObj:=wPaper;
    MoveL Offs(pOrigin,340.51,285.14,0.00),v40,fine,tPen\WObj:=wPaper;
    MoveL Offs(pOrigin,340.51,285.14,6.00),v60,z5,tPen\WObj:=wPaper;
    MoveL Offs(pOrigin,338.11,288.01,6.00),vTravel,z5,tPen\WObj:=wPaper;
    MoveL Offs(pOrigin,338.11,288.01,0.00),v60,z0,tPen\WObj:=wPaper;
    MoveL Offs(pOrigin,338.11,288.49,0.00),v40,z0,tPen\WObj:=wPaper;
    MoveL Offs(pOrigin,337.63,288.49,0.00),v40,z0,tPen\WObj:=wPaper;
    MoveL Offs(pOrigin,337.15,288.97,0.00),v40,z0,tPen\WObj:=wPaper;
    MoveL Offs(pOrigin,338.11,288.01,0.00),v40,z0,tPen\WObj:=wPaper;
    MoveL Offs(pOrigin,338.11,288.49,0.00),v40,z0,tPen\WObj:=wPaper;
    MoveL Offs(pOrigin,337.63,288.49,0.00),v40,z0,tPen\WObj:=wPaper;
    MoveL Offs(pOrigin,337.15,288.97,0.00),v40,z0,tPen\WObj:=wPaper;
    MoveL Offs(pOrigin,338.11,288.01,0.00),v40,fine,tPen\WObj:=wPaper;
    MoveL Offs(pOrigin,338.11,288.01,6.00),v60,z5,tPen\WObj:=wPaper;
    MoveL Offs(pOrigin,336.68,289.45,6.00),vTravel,z5,tPen\WObj:=wPaper;
    MoveL Offs(pOrigin,336.68,289.45,0.00),v60,z0,tPen\WObj:=wPaper;
    MoveL Offs(pOrigin,336.68,289.93,0.00),v40,z0,tPen\WObj:=wPaper;
    MoveL Offs(pOrigin,336.20,289.93,0.00),v40,z0,tPen\WObj:=wPaper;
    MoveL Offs(pOrigin,334.28,291.85,0.00),v40,z0,tPen\WObj:=wPaper;
    MoveL Offs(pOrigin,336.68,289.45,0.00),v40,z0,tPen\WObj:=wPaper;
    MoveL Offs(pOrigin,336.68,289.93,0.00),v40,z0,tPen\WObj:=wPaper;
    MoveL Offs(pOrigin,336.20,289.93,0.00),v40,z0,tPen\WObj:=wPaper;
    MoveL Offs(pOrigin,334.28,291.85,0.00),v40,z0,tPen\WObj:=wPaper;
    MoveL Offs(pOrigin,336.68,289.45,0.00),v40,fine,tPen\WObj:=wPaper;
    MoveL Offs(pOrigin,336.68,289.45,6.00),v60,z5,tPen\WObj:=wPaper;
    MoveL Offs(pOrigin,333.80,292.32,6.00),vTravel,z5,tPen\WObj:=wPaper;
    MoveL Offs(pOrigin,333.80,292.32,0.00),v60,z0,tPen\WObj:=wPaper;
    MoveL Offs(pOrigin,333.80,292.80,0.00),v40,z0,tPen\WObj:=wPaper;
    MoveL Offs(pOrigin,333.32,292.80,0.00),v40,z0,tPen\WObj:=wPaper;
    MoveL Offs(pOrigin,332.85,293.28,0.00),v40,z0,tPen\WObj:=wPaper;
    MoveL Offs(pOrigin,333.80,292.32,0.00),v40,z0,tPen\WObj:=wPaper;
    MoveL Offs(pOrigin,333.80,292.80,0.00),v40,z0,tPen\WObj:=wPaper;
    MoveL Offs(pOrigin,333.32,292.80,0.00),v40,z0,tPen\WObj:=wPaper;
    MoveL Offs(pOrigin,332.85,293.28,0.00),v40,z0,tPen\WObj:=wPaper;
    MoveL Offs(pOrigin,333.80,292.32,0.00),v40,fine,tPen\WObj:=wPaper;
    MoveL Offs(pOrigin,333.80,292.32,6.00),v60,z5,tPen\WObj:=wPaper;
    MoveL Offs(pOrigin,332.21,294.08,6.00),vTravel,z5,tPen\WObj:=wPaper;
    MoveL Offs(pOrigin,332.21,294.08,0.00),v60,z0,tPen\WObj:=wPaper;
    MoveL Offs(pOrigin,327.58,298.55,0.00),v40,z0,tPen\WObj:=wPaper;
    MoveL Offs(pOrigin,332.21,294.08,0.00),v40,fine,tPen\WObj:=wPaper;
    MoveL Offs(pOrigin,332.21,294.08,6.00),v60,z5,tPen\WObj:=wPaper;
    MoveL Offs(pOrigin,328.22,283.86,6.00),vTravel,z5,tPen\WObj:=wPaper;
    MoveL Offs(pOrigin,328.22,283.86,0.00),v60,z0,tPen\WObj:=wPaper;
    MoveL Offs(pOrigin,334.28,275.08,0.00),v40,z0,tPen\WObj:=wPaper;
    MoveL Offs(pOrigin,334.12,277.00,0.00),v40,z0,tPen\WObj:=wPaper;
    MoveL Offs(pOrigin,332.69,279.87,0.00),v40,z0,tPen\WObj:=wPaper;
    MoveL Offs(pOrigin,329.49,283.07,0.00),v40,z0,tPen\WObj:=wPaper;
    MoveL Offs(pOrigin,328.54,283.38,0.00),v40,z0,tPen\WObj:=wPaper;
    MoveL Offs(pOrigin,328.22,283.86,0.00),v40,fine,tPen\WObj:=wPaper;
    MoveL Offs(pOrigin,328.22,283.86,6.00),v60,z5,tPen\WObj:=wPaper;
    MoveL Offs(pOrigin,330.45,282.27,6.00),vTravel,z5,tPen\WObj:=wPaper;
    MoveL Offs(pOrigin,330.45,282.27,0.00),v60,z0,tPen\WObj:=wPaper;
    MoveL Offs(pOrigin,330.93,281.79,0.00),v40,z0,tPen\WObj:=wPaper;
    MoveL Offs(pOrigin,330.93,281.31,0.00),v40,z0,tPen\WObj:=wPaper;
    MoveL Offs(pOrigin,330.45,282.27,0.00),v40,z0,tPen\WObj:=wPaper;
    MoveL Offs(pOrigin,330.93,281.79,0.00),v40,z0,tPen\WObj:=wPaper;
    MoveL Offs(pOrigin,330.93,281.31,0.00),v40,z0,tPen\WObj:=wPaper;
    MoveL Offs(pOrigin,330.45,282.27,0.00),v40,fine,tPen\WObj:=wPaper;
    MoveL Offs(pOrigin,330.45,282.27,6.00),v60,z5,tPen\WObj:=wPaper;
    MoveL Offs(pOrigin,331.89,280.83,6.00),vTravel,z5,tPen\WObj:=wPaper;
    MoveL Offs(pOrigin,331.89,280.83,0.00),v60,z0,tPen\WObj:=wPaper;
    MoveL Offs(pOrigin,332.37,280.35,0.00),v40,z0,tPen\WObj:=wPaper;
    MoveL Offs(pOrigin,332.37,279.87,0.00),v40,z0,tPen\WObj:=wPaper;
    MoveL Offs(pOrigin,331.89,280.83,0.00),v40,z0,tPen\WObj:=wPaper;
    MoveL Offs(pOrigin,332.37,280.35,0.00),v40,z0,tPen\WObj:=wPaper;
    MoveL Offs(pOrigin,332.37,279.87,0.00),v40,z0,tPen\WObj:=wPaper;
    MoveL Offs(pOrigin,331.89,280.83,0.00),v40,fine,tPen\WObj:=wPaper;
    MoveL Offs(pOrigin,331.89,280.83,6.00),v60,z5,tPen\WObj:=wPaper;
    MoveL Offs(pOrigin,334.28,273.65,6.00),vTravel,z5,tPen\WObj:=wPaper;
    MoveL Offs(pOrigin,334.28,273.65,0.00),v60,z0,tPen\WObj:=wPaper;
    MoveL Offs(pOrigin,330.93,265.51,0.00),v40,z0,tPen\WObj:=wPaper;
    MoveL Offs(pOrigin,333.00,268.38,0.00),v40,z0,tPen\WObj:=wPaper;
    MoveL Offs(pOrigin,334.12,270.77,0.00),v40,z0,tPen\WObj:=wPaper;
    MoveL Offs(pOrigin,334.28,273.65,0.00),v40,fine,tPen\WObj:=wPaper;
    MoveL Offs(pOrigin,334.28,273.65,6.00),v60,z5,tPen\WObj:=wPaper;
    MoveL Offs(pOrigin,328.06,263.11,6.00),vTravel,z5,tPen\WObj:=wPaper;
    MoveL Offs(pOrigin,328.06,263.11,0.00),v60,z0,tPen\WObj:=wPaper;
    MoveL Offs(pOrigin,327.58,262.63,0.00),v40,z0,tPen\WObj:=wPaper;
    MoveL Offs(pOrigin,327.58,263.11,0.00),v40,z0,tPen\WObj:=wPaper;
    MoveL Offs(pOrigin,328.06,263.11,0.00),v40,z0,tPen\WObj:=wPaper;
    MoveL Offs(pOrigin,327.58,262.63,0.00),v40,z0,tPen\WObj:=wPaper;
    MoveL Offs(pOrigin,327.58,263.11,0.00),v40,z0,tPen\WObj:=wPaper;
    MoveL Offs(pOrigin,328.06,263.11,0.00),v40,fine,tPen\WObj:=wPaper;
    MoveL Offs(pOrigin,328.06,263.11,6.00),v60,z5,tPen\WObj:=wPaper;
    MoveL Offs(pOrigin,340.51,263.11,6.00),vTravel,z5,tPen\WObj:=wPaper;
    MoveL Offs(pOrigin,340.51,263.11,0.00),v60,z0,tPen\WObj:=wPaper;
    MoveL Offs(pOrigin,340.99,263.11,0.00),v40,z0,tPen\WObj:=wPaper;
    MoveL Offs(pOrigin,341.46,263.59,0.00),v40,z0,tPen\WObj:=wPaper;
    MoveL Offs(pOrigin,340.51,263.11,0.00),v40,z0,tPen\WObj:=wPaper;
    MoveL Offs(pOrigin,340.99,263.11,0.00),v40,z0,tPen\WObj:=wPaper;
    MoveL Offs(pOrigin,341.46,263.59,0.00),v40,z0,tPen\WObj:=wPaper;
    MoveL Offs(pOrigin,340.51,263.11,0.00),v40,fine,tPen\WObj:=wPaper;
    MoveL Offs(pOrigin,340.51,263.11,6.00),v60,z5,tPen\WObj:=wPaper;
  ENDPROC

  PROC DrawPart28()
    MoveL Offs(pOrigin,344.34,255.93,6.00),vTravel,z5,tPen\WObj:=wPaper;
    MoveL Offs(pOrigin,344.34,255.93,0.00),v60,z0,tPen\WObj:=wPaper;
    MoveL Offs(pOrigin,344.82,255.93,0.00),v40,z0,tPen\WObj:=wPaper;
    MoveL Offs(pOrigin,344.34,255.45,0.00),v40,z0,tPen\WObj:=wPaper;
    MoveL Offs(pOrigin,344.34,255.93,0.00),v40,z0,tPen\WObj:=wPaper;
    MoveL Offs(pOrigin,344.82,255.93,0.00),v40,z0,tPen\WObj:=wPaper;
    MoveL Offs(pOrigin,344.34,255.45,0.00),v40,z0,tPen\WObj:=wPaper;
    MoveL Offs(pOrigin,344.34,255.93,0.00),v40,fine,tPen\WObj:=wPaper;
    MoveL Offs(pOrigin,344.34,255.93,6.00),v60,z5,tPen\WObj:=wPaper;
    MoveL Offs(pOrigin,355.83,245.87,6.00),vTravel,z5,tPen\WObj:=wPaper;
    MoveL Offs(pOrigin,355.83,245.87,0.00),v60,z0,tPen\WObj:=wPaper;
    MoveL Offs(pOrigin,356.79,246.83,0.00),v40,z0,tPen\WObj:=wPaper;
    MoveL Offs(pOrigin,355.83,245.87,0.00),v40,z0,tPen\WObj:=wPaper;
    MoveL Offs(pOrigin,356.31,245.87,0.00),v40,z0,tPen\WObj:=wPaper;
    MoveL Offs(pOrigin,355.83,244.92,0.00),v40,z0,tPen\WObj:=wPaper;
    MoveL Offs(pOrigin,359.98,235.34,0.00),v40,z0,tPen\WObj:=wPaper;
    MoveL Offs(pOrigin,362.06,229.11,0.00),v40,z0,tPen\WObj:=wPaper;
    MoveL Offs(pOrigin,365.41,216.18,0.00),v40,z0,tPen\WObj:=wPaper;
    MoveL Offs(pOrigin,365.41,213.79,0.00),v40,z0,tPen\WObj:=wPaper;
    MoveL Offs(pOrigin,366.37,209.96,0.00),v40,z0,tPen\WObj:=wPaper;
    MoveL Offs(pOrigin,366.37,206.13,0.00),v40,z0,tPen\WObj:=wPaper;
    MoveL Offs(pOrigin,367.00,203.73,0.00),v40,z0,tPen\WObj:=wPaper;
    MoveL Offs(pOrigin,368.28,202.77,0.00),v40,z0,tPen\WObj:=wPaper;
    MoveL Offs(pOrigin,372.59,203.89,0.00),v40,z0,tPen\WObj:=wPaper;
    MoveL Offs(pOrigin,373.55,205.17,0.00),v40,z0,tPen\WObj:=wPaper;
    MoveL Offs(pOrigin,373.55,209.48,0.00),v40,z0,tPen\WObj:=wPaper;
    MoveL Offs(pOrigin,372.59,213.79,0.00),v40,z0,tPen\WObj:=wPaper;
    MoveL Offs(pOrigin,372.59,217.14,0.00),v40,z0,tPen\WObj:=wPaper;
    MoveL Offs(pOrigin,369.72,229.59,0.00),v40,z0,tPen\WObj:=wPaper;
    MoveL Offs(pOrigin,366.05,240.61,0.00),v40,z0,tPen\WObj:=wPaper;
    MoveL Offs(pOrigin,362.85,247.79,0.00),v40,z0,tPen\WObj:=wPaper;
    MoveL Offs(pOrigin,362.06,248.27,0.00),v40,z0,tPen\WObj:=wPaper;
    MoveL Offs(pOrigin,361.10,248.27,0.00),v40,z0,tPen\WObj:=wPaper;
    MoveL Offs(pOrigin,357.75,246.99,0.00),v40,z0,tPen\WObj:=wPaper;
    MoveL Offs(pOrigin,356.31,245.87,0.00),v40,fine,tPen\WObj:=wPaper;
    MoveL Offs(pOrigin,356.31,245.87,6.00),v60,z5,tPen\WObj:=wPaper;
    MoveL Offs(pOrigin,355.83,243.96,6.00),vTravel,z5,tPen\WObj:=wPaper;
    MoveL Offs(pOrigin,355.83,243.96,0.00),v60,z0,tPen\WObj:=wPaper;
    MoveL Offs(pOrigin,356.31,243.00,0.00),v40,z0,tPen\WObj:=wPaper;
    MoveL Offs(pOrigin,356.31,243.48,0.00),v40,z0,tPen\WObj:=wPaper;
    MoveL Offs(pOrigin,355.83,243.96,0.00),v40,z0,tPen\WObj:=wPaper;
    MoveL Offs(pOrigin,356.31,243.00,0.00),v40,z0,tPen\WObj:=wPaper;
    MoveL Offs(pOrigin,356.31,243.48,0.00),v40,z0,tPen\WObj:=wPaper;
    MoveL Offs(pOrigin,355.83,243.96,0.00),v40,fine,tPen\WObj:=wPaper;
    MoveL Offs(pOrigin,355.83,243.96,6.00),v60,z5,tPen\WObj:=wPaper;
    MoveL Offs(pOrigin,345.77,221.61,6.00),vTravel,z5,tPen\WObj:=wPaper;
    MoveL Offs(pOrigin,345.77,221.61,0.00),v60,z0,tPen\WObj:=wPaper;
    MoveL Offs(pOrigin,347.69,220.49,0.00),v40,z0,tPen\WObj:=wPaper;
    MoveL Offs(pOrigin,349.29,218.58,0.00),v40,z0,tPen\WObj:=wPaper;
    MoveL Offs(pOrigin,350.08,214.75,0.00),v40,z0,tPen\WObj:=wPaper;
    MoveL Offs(pOrigin,349.13,212.35,0.00),v40,z0,tPen\WObj:=wPaper;
    MoveL Offs(pOrigin,346.25,209.48,0.00),v40,z0,tPen\WObj:=wPaper;
    MoveL Offs(pOrigin,342.74,204.69,0.00),v40,z0,tPen\WObj:=wPaper;
    MoveL Offs(pOrigin,341.46,201.34,0.00),v40,z0,tPen\WObj:=wPaper;
    MoveL Offs(pOrigin,341.46,198.94,0.00),v40,z0,tPen\WObj:=wPaper;
    MoveL Offs(pOrigin,341.78,197.99,0.00),v40,z0,tPen\WObj:=wPaper;
    MoveL Offs(pOrigin,344.34,193.68,0.00),v40,z0,tPen\WObj:=wPaper;
    MoveL Offs(pOrigin,351.68,184.10,0.00),v40,z0,tPen\WObj:=wPaper;
    MoveL Offs(pOrigin,352.48,183.62,0.00),v40,z0,tPen\WObj:=wPaper;
    MoveL Offs(pOrigin,353.92,183.62,0.00),v40,z0,tPen\WObj:=wPaper;
    MoveL Offs(pOrigin,358.23,185.22,0.00),v40,z0,tPen\WObj:=wPaper;
    MoveL Offs(pOrigin,362.06,187.45,0.00),v40,z0,tPen\WObj:=wPaper;
    MoveL Offs(pOrigin,364.93,190.32,0.00),v40,z0,tPen\WObj:=wPaper;
    MoveL Offs(pOrigin,367.32,191.76,0.00),v40,z0,tPen\WObj:=wPaper;
    MoveL Offs(pOrigin,370.68,191.76,0.00),v40,z0,tPen\WObj:=wPaper;
    MoveL Offs(pOrigin,372.59,190.80,0.00),v40,z0,tPen\WObj:=wPaper;
    MoveL Offs(pOrigin,374.03,187.45,0.00),v40,z0,tPen\WObj:=wPaper;
    MoveL Offs(pOrigin,374.03,186.01,0.00),v40,z0,tPen\WObj:=wPaper;
    MoveL Offs(pOrigin,373.39,184.10,0.00),v40,z0,tPen\WObj:=wPaper;
    MoveL Offs(pOrigin,370.68,179.79,0.00),v40,z0,tPen\WObj:=wPaper;
    MoveL Offs(pOrigin,369.72,178.83,0.00),v40,z0,tPen\WObj:=wPaper;
    MoveL Offs(pOrigin,364.45,175.32,0.00),v40,z0,tPen\WObj:=wPaper;
    MoveL Offs(pOrigin,357.27,172.45,0.00),v40,z0,tPen\WObj:=wPaper;
    MoveL Offs(pOrigin,356.31,171.65,0.00),v40,z0,tPen\WObj:=wPaper;
    MoveL Offs(pOrigin,355.83,170.69,0.00),v40,z0,tPen\WObj:=wPaper;
    MoveL Offs(pOrigin,355.83,167.82,0.00),v40,z0,tPen\WObj:=wPaper;
    MoveL Offs(pOrigin,354.39,161.59,0.00),v40,z0,tPen\WObj:=wPaper;
    MoveL Offs(pOrigin,351.84,155.85,0.00),v40,z0,tPen\WObj:=wPaper;
    MoveL Offs(pOrigin,349.61,152.49,0.00),v40,z0,tPen\WObj:=wPaper;
    MoveL Offs(pOrigin,343.38,146.27,0.00),v40,z0,tPen\WObj:=wPaper;
    MoveL Offs(pOrigin,339.55,143.71,0.00),v40,z0,tPen\WObj:=wPaper;
    MoveL Offs(pOrigin,332.37,140.52,0.00),v40,z0,tPen\WObj:=wPaper;
    MoveL Offs(pOrigin,331.41,140.52,0.00),v40,z0,tPen\WObj:=wPaper;
    MoveL Offs(pOrigin,326.14,139.08,0.00),v40,z0,tPen\WObj:=wPaper;
    MoveL Offs(pOrigin,323.27,139.08,0.00),v40,z0,tPen\WObj:=wPaper;
    MoveL Offs(pOrigin,321.83,138.61,0.00),v40,z0,tPen\WObj:=wPaper;
    MoveL Offs(pOrigin,317.52,138.61,0.00),v40,z0,tPen\WObj:=wPaper;
    MoveL Offs(pOrigin,316.08,139.08,0.00),v40,z0,tPen\WObj:=wPaper;
    MoveL Offs(pOrigin,313.21,139.08,0.00),v40,z0,tPen\WObj:=wPaper;
    MoveL Offs(pOrigin,306.51,141.32,0.00),v40,z0,tPen\WObj:=wPaper;
    MoveL Offs(pOrigin,305.71,142.12,0.00),v40,z0,tPen\WObj:=wPaper;
    MoveL Offs(pOrigin,333.32,220.97,0.00),v40,z0,tPen\WObj:=wPaper;
    MoveL Offs(pOrigin,335.72,221.93,0.00),v40,z0,tPen\WObj:=wPaper;
    MoveL Offs(pOrigin,338.11,222.41,0.00),v40,z0,tPen\WObj:=wPaper;
    MoveL Offs(pOrigin,342.90,222.41,0.00),v40,z0,tPen\WObj:=wPaper;
    MoveL Offs(pOrigin,345.77,221.61,0.00),v40,fine,tPen\WObj:=wPaper;
    MoveL Offs(pOrigin,345.77,221.61,6.00),v60,z5,tPen\WObj:=wPaper;
    MoveL Offs(pOrigin,347.21,220.49,6.00),vTravel,z5,tPen\WObj:=wPaper;
    MoveL Offs(pOrigin,347.21,220.49,0.00),v60,z0,tPen\WObj:=wPaper;
    MoveL Offs(pOrigin,347.69,220.01,0.00),v40,z0,tPen\WObj:=wPaper;
    MoveL Offs(pOrigin,347.69,220.49,0.00),v40,z0,tPen\WObj:=wPaper;
    MoveL Offs(pOrigin,347.21,220.49,0.00),v40,z0,tPen\WObj:=wPaper;
    MoveL Offs(pOrigin,347.69,220.01,0.00),v40,z0,tPen\WObj:=wPaper;
    MoveL Offs(pOrigin,347.69,220.49,0.00),v40,z0,tPen\WObj:=wPaper;
    MoveL Offs(pOrigin,347.21,220.49,0.00),v40,fine,tPen\WObj:=wPaper;
    MoveL Offs(pOrigin,347.21,220.49,6.00),v60,z5,tPen\WObj:=wPaper;
    MoveL Offs(pOrigin,348.17,219.54,6.00),vTravel,z5,tPen\WObj:=wPaper;
    MoveL Offs(pOrigin,348.17,219.54,0.00),v60,z0,tPen\WObj:=wPaper;
    MoveL Offs(pOrigin,349.13,218.10,0.00),v40,z0,tPen\WObj:=wPaper;
    MoveL Offs(pOrigin,349.13,218.58,0.00),v40,z0,tPen\WObj:=wPaper;
    MoveL Offs(pOrigin,348.17,219.54,0.00),v40,z0,tPen\WObj:=wPaper;
    MoveL Offs(pOrigin,349.13,218.10,0.00),v40,z0,tPen\WObj:=wPaper;
    MoveL Offs(pOrigin,349.13,218.58,0.00),v40,z0,tPen\WObj:=wPaper;
    MoveL Offs(pOrigin,348.17,219.54,0.00),v40,fine,tPen\WObj:=wPaper;
    MoveL Offs(pOrigin,348.17,219.54,6.00),v60,z5,tPen\WObj:=wPaper;
    MoveL Offs(pOrigin,346.25,209.96,6.00),vTravel,z5,tPen\WObj:=wPaper;
    MoveL Offs(pOrigin,346.25,209.96,0.00),v60,z0,tPen\WObj:=wPaper;
    MoveL Offs(pOrigin,349.13,212.83,0.00),v40,z0,tPen\WObj:=wPaper;
    MoveL Offs(pOrigin,346.25,209.96,0.00),v40,fine,tPen\WObj:=wPaper;
    MoveL Offs(pOrigin,346.25,209.96,6.00),v60,z5,tPen\WObj:=wPaper;
  ENDPROC

  PROC DrawPart29()
    MoveL Offs(pOrigin,344.34,207.56,6.00),vTravel,z5,tPen\WObj:=wPaper;
    MoveL Offs(pOrigin,344.34,207.56,0.00),v60,z0,tPen\WObj:=wPaper;
    MoveL Offs(pOrigin,345.30,208.52,0.00),v40,z0,tPen\WObj:=wPaper;
    MoveL Offs(pOrigin,344.34,207.56,0.00),v40,fine,tPen\WObj:=wPaper;
    MoveL Offs(pOrigin,344.34,207.56,6.00),v60,z5,tPen\WObj:=wPaper;
    MoveL Offs(pOrigin,344.34,193.68,6.00),vTravel,z5,tPen\WObj:=wPaper;
    MoveL Offs(pOrigin,344.34,193.68,0.00),v60,z0,tPen\WObj:=wPaper;
    MoveL Offs(pOrigin,343.86,193.68,0.00),v40,z0,tPen\WObj:=wPaper;
    MoveL Offs(pOrigin,344.34,193.20,0.00),v40,z0,tPen\WObj:=wPaper;
    MoveL Offs(pOrigin,344.34,193.68,0.00),v40,z0,tPen\WObj:=wPaper;
    MoveL Offs(pOrigin,343.86,193.68,0.00),v40,z0,tPen\WObj:=wPaper;
    MoveL Offs(pOrigin,344.34,193.20,0.00),v40,z0,tPen\WObj:=wPaper;
    MoveL Offs(pOrigin,344.34,193.68,0.00),v40,fine,tPen\WObj:=wPaper;
    MoveL Offs(pOrigin,344.34,193.68,6.00),v60,z5,tPen\WObj:=wPaper;
    MoveL Offs(pOrigin,345.30,191.76,6.00),vTravel,z5,tPen\WObj:=wPaper;
    MoveL Offs(pOrigin,345.30,191.76,0.00),v60,z0,tPen\WObj:=wPaper;
    MoveL Offs(pOrigin,347.21,189.37,0.00),v40,z0,tPen\WObj:=wPaper;
    MoveL Offs(pOrigin,347.21,189.85,0.00),v40,z0,tPen\WObj:=wPaper;
    MoveL Offs(pOrigin,345.30,191.76,0.00),v40,z0,tPen\WObj:=wPaper;
    MoveL Offs(pOrigin,347.21,189.37,0.00),v40,z0,tPen\WObj:=wPaper;
    MoveL Offs(pOrigin,347.21,189.85,0.00),v40,z0,tPen\WObj:=wPaper;
    MoveL Offs(pOrigin,345.30,191.76,0.00),v40,fine,tPen\WObj:=wPaper;
    MoveL Offs(pOrigin,345.30,191.76,6.00),v60,z5,tPen\WObj:=wPaper;
    MoveL Offs(pOrigin,348.65,187.45,6.00),vTravel,z5,tPen\WObj:=wPaper;
    MoveL Offs(pOrigin,348.65,187.45,0.00),v60,z0,tPen\WObj:=wPaper;
    MoveL Offs(pOrigin,350.08,185.54,0.00),v40,z0,tPen\WObj:=wPaper;
    MoveL Offs(pOrigin,350.08,186.01,0.00),v40,z0,tPen\WObj:=wPaper;
    MoveL Offs(pOrigin,348.65,187.45,0.00),v40,z0,tPen\WObj:=wPaper;
    MoveL Offs(pOrigin,350.08,185.54,0.00),v40,z0,tPen\WObj:=wPaper;
    MoveL Offs(pOrigin,350.08,186.01,0.00),v40,z0,tPen\WObj:=wPaper;
    MoveL Offs(pOrigin,348.65,187.45,0.00),v40,fine,tPen\WObj:=wPaper;
    MoveL Offs(pOrigin,348.65,187.45,6.00),v60,z5,tPen\WObj:=wPaper;
    MoveL Offs(pOrigin,362.54,187.45,6.00),vTravel,z5,tPen\WObj:=wPaper;
    MoveL Offs(pOrigin,362.54,187.45,0.00),v60,z0,tPen\WObj:=wPaper;
    MoveL Offs(pOrigin,362.54,187.93,0.00),v40,z0,tPen\WObj:=wPaper;
    MoveL Offs(pOrigin,363.01,187.93,0.00),v40,z0,tPen\WObj:=wPaper;
    MoveL Offs(pOrigin,365.41,190.32,0.00),v40,z0,tPen\WObj:=wPaper;
    MoveL Offs(pOrigin,362.54,187.45,0.00),v40,z0,tPen\WObj:=wPaper;
    MoveL Offs(pOrigin,362.54,187.93,0.00),v40,z0,tPen\WObj:=wPaper;
    MoveL Offs(pOrigin,363.01,187.93,0.00),v40,z0,tPen\WObj:=wPaper;
    MoveL Offs(pOrigin,365.41,190.32,0.00),v40,z0,tPen\WObj:=wPaper;
    MoveL Offs(pOrigin,362.54,187.45,0.00),v40,fine,tPen\WObj:=wPaper;
    MoveL Offs(pOrigin,362.54,187.45,6.00),v60,z5,tPen\WObj:=wPaper;
    MoveL Offs(pOrigin,372.11,190.80,6.00),vTravel,z5,tPen\WObj:=wPaper;
    MoveL Offs(pOrigin,372.11,190.80,0.00),v60,z0,tPen\WObj:=wPaper;
    MoveL Offs(pOrigin,373.07,189.37,0.00),v40,z0,tPen\WObj:=wPaper;
    MoveL Offs(pOrigin,373.07,189.85,0.00),v40,z0,tPen\WObj:=wPaper;
    MoveL Offs(pOrigin,372.11,190.80,0.00),v40,z0,tPen\WObj:=wPaper;
    MoveL Offs(pOrigin,373.07,189.37,0.00),v40,z0,tPen\WObj:=wPaper;
    MoveL Offs(pOrigin,373.07,189.85,0.00),v40,z0,tPen\WObj:=wPaper;
    MoveL Offs(pOrigin,372.11,190.80,0.00),v40,fine,tPen\WObj:=wPaper;
    MoveL Offs(pOrigin,372.11,190.80,6.00),v60,z5,tPen\WObj:=wPaper;
    MoveL Offs(pOrigin,370.68,180.27,6.00),vTravel,z5,tPen\WObj:=wPaper;
    MoveL Offs(pOrigin,370.68,180.27,0.00),v60,z0,tPen\WObj:=wPaper;
    MoveL Offs(pOrigin,368.28,178.35,0.00),v40,z0,tPen\WObj:=wPaper;
    MoveL Offs(pOrigin,368.76,178.35,0.00),v40,z0,tPen\WObj:=wPaper;
    MoveL Offs(pOrigin,370.68,180.27,0.00),v40,z0,tPen\WObj:=wPaper;
    MoveL Offs(pOrigin,368.28,178.35,0.00),v40,z0,tPen\WObj:=wPaper;
    MoveL Offs(pOrigin,368.76,178.35,0.00),v40,z0,tPen\WObj:=wPaper;
    MoveL Offs(pOrigin,370.68,180.27,0.00),v40,fine,tPen\WObj:=wPaper;
    MoveL Offs(pOrigin,370.68,180.27,6.00),v60,z5,tPen\WObj:=wPaper;
    MoveL Offs(pOrigin,367.80,177.87,6.00),vTravel,z5,tPen\WObj:=wPaper;
    MoveL Offs(pOrigin,367.80,177.87,0.00),v60,z0,tPen\WObj:=wPaper;
    MoveL Offs(pOrigin,366.85,177.39,0.00),v40,z0,tPen\WObj:=wPaper;
    MoveL Offs(pOrigin,367.32,177.39,0.00),v40,z0,tPen\WObj:=wPaper;
    MoveL Offs(pOrigin,367.80,177.87,0.00),v40,z0,tPen\WObj:=wPaper;
    MoveL Offs(pOrigin,366.85,177.39,0.00),v40,z0,tPen\WObj:=wPaper;
    MoveL Offs(pOrigin,367.32,177.39,0.00),v40,z0,tPen\WObj:=wPaper;
    MoveL Offs(pOrigin,367.80,177.87,0.00),v40,fine,tPen\WObj:=wPaper;
    MoveL Offs(pOrigin,367.80,177.87,6.00),v60,z5,tPen\WObj:=wPaper;
    MoveL Offs(pOrigin,364.45,157.76,6.00),vTravel,z5,tPen\WObj:=wPaper;
    MoveL Offs(pOrigin,364.45,157.76,0.00),v60,z0,tPen\WObj:=wPaper;
    MoveL Offs(pOrigin,366.85,160.15,0.00),v40,z0,tPen\WObj:=wPaper;
    MoveL Offs(pOrigin,364.45,157.76,0.00),v40,fine,tPen\WObj:=wPaper;
    MoveL Offs(pOrigin,364.45,157.76,6.00),v60,z5,tPen\WObj:=wPaper;
    MoveL Offs(pOrigin,361.58,155.37,6.00),vTravel,z5,tPen\WObj:=wPaper;
    MoveL Offs(pOrigin,361.58,155.37,0.00),v60,z0,tPen\WObj:=wPaper;
    MoveL Offs(pOrigin,363.01,156.80,0.00),v40,z0,tPen\WObj:=wPaper;
    MoveL Offs(pOrigin,361.58,155.37,0.00),v40,fine,tPen\WObj:=wPaper;
    MoveL Offs(pOrigin,361.58,155.37,6.00),v60,z5,tPen\WObj:=wPaper;
    MoveL Offs(pOrigin,359.66,153.45,6.00),vTravel,z5,tPen\WObj:=wPaper;
    MoveL Offs(pOrigin,359.66,153.45,0.00),v60,z0,tPen\WObj:=wPaper;
    MoveL Offs(pOrigin,361.10,154.89,0.00),v40,z0,tPen\WObj:=wPaper;
    MoveL Offs(pOrigin,359.66,153.45,0.00),v40,fine,tPen\WObj:=wPaper;
    MoveL Offs(pOrigin,359.66,153.45,6.00),v60,z5,tPen\WObj:=wPaper;
    MoveL Offs(pOrigin,352.96,158.24,6.00),vTravel,z5,tPen\WObj:=wPaper;
    MoveL Offs(pOrigin,352.96,158.24,0.00),v60,z0,tPen\WObj:=wPaper;
    MoveL Offs(pOrigin,352.96,158.72,0.00),v40,z0,tPen\WObj:=wPaper;
    MoveL Offs(pOrigin,352.48,157.76,0.00),v40,z0,tPen\WObj:=wPaper;
    MoveL Offs(pOrigin,352.96,158.24,0.00),v40,z0,tPen\WObj:=wPaper;
    MoveL Offs(pOrigin,352.96,158.72,0.00),v40,z0,tPen\WObj:=wPaper;
    MoveL Offs(pOrigin,352.48,157.76,0.00),v40,z0,tPen\WObj:=wPaper;
    MoveL Offs(pOrigin,352.96,158.24,0.00),v40,fine,tPen\WObj:=wPaper;
    MoveL Offs(pOrigin,352.96,158.24,6.00),v60,z5,tPen\WObj:=wPaper;
    MoveL Offs(pOrigin,351.04,155.37,6.00),vTravel,z5,tPen\WObj:=wPaper;
    MoveL Offs(pOrigin,351.04,155.37,0.00),v60,z0,tPen\WObj:=wPaper;
    MoveL Offs(pOrigin,350.56,154.41,0.00),v40,z0,tPen\WObj:=wPaper;
    MoveL Offs(pOrigin,351.04,154.89,0.00),v40,z0,tPen\WObj:=wPaper;
    MoveL Offs(pOrigin,351.04,155.37,0.00),v40,z0,tPen\WObj:=wPaper;
    MoveL Offs(pOrigin,350.56,154.41,0.00),v40,z0,tPen\WObj:=wPaper;
    MoveL Offs(pOrigin,351.04,154.89,0.00),v40,z0,tPen\WObj:=wPaper;
    MoveL Offs(pOrigin,351.04,155.37,0.00),v40,fine,tPen\WObj:=wPaper;
    MoveL Offs(pOrigin,351.04,155.37,6.00),v60,z5,tPen\WObj:=wPaper;
    MoveL Offs(pOrigin,345.77,149.14,6.00),vTravel,z5,tPen\WObj:=wPaper;
    MoveL Offs(pOrigin,345.77,149.14,0.00),v60,z0,tPen\WObj:=wPaper;
    MoveL Offs(pOrigin,349.61,152.97,0.00),v40,z0,tPen\WObj:=wPaper;
    MoveL Offs(pOrigin,345.77,149.14,0.00),v40,fine,tPen\WObj:=wPaper;
    MoveL Offs(pOrigin,345.77,149.14,6.00),v60,z5,tPen\WObj:=wPaper;
    MoveL Offs(pOrigin,343.86,147.23,6.00),vTravel,z5,tPen\WObj:=wPaper;
    MoveL Offs(pOrigin,343.86,147.23,0.00),v60,z0,tPen\WObj:=wPaper;
    MoveL Offs(pOrigin,344.82,148.18,0.00),v40,z0,tPen\WObj:=wPaper;
    MoveL Offs(pOrigin,343.86,147.23,0.00),v40,z0,tPen\WObj:=wPaper;
    MoveL Offs(pOrigin,343.38,146.75,0.00),v40,z0,tPen\WObj:=wPaper;
    MoveL Offs(pOrigin,341.94,145.79,0.00),v40,z0,tPen\WObj:=wPaper;
    MoveL Offs(pOrigin,342.42,145.79,0.00),v40,z0,tPen\WObj:=wPaper;
    MoveL Offs(pOrigin,343.38,146.75,0.00),v40,z0,tPen\WObj:=wPaper;
    MoveL Offs(pOrigin,341.94,145.79,0.00),v40,z0,tPen\WObj:=wPaper;
    MoveL Offs(pOrigin,342.42,145.79,0.00),v40,z0,tPen\WObj:=wPaper;
    MoveL Offs(pOrigin,343.38,146.75,0.00),v40,fine,tPen\WObj:=wPaper;
    MoveL Offs(pOrigin,343.38,146.75,6.00),v60,z5,tPen\WObj:=wPaper;
  ENDPROC

  PROC DrawPart30()
    MoveL Offs(pOrigin,339.07,143.87,6.00),vTravel,z5,tPen\WObj:=wPaper;
    MoveL Offs(pOrigin,339.07,143.87,0.00),v60,z0,tPen\WObj:=wPaper;
    MoveL Offs(pOrigin,338.11,143.39,0.00),v40,z0,tPen\WObj:=wPaper;
    MoveL Offs(pOrigin,338.59,143.39,0.00),v40,z0,tPen\WObj:=wPaper;
    MoveL Offs(pOrigin,339.07,143.87,0.00),v40,z0,tPen\WObj:=wPaper;
    MoveL Offs(pOrigin,338.11,143.39,0.00),v40,z0,tPen\WObj:=wPaper;
    MoveL Offs(pOrigin,338.59,143.39,0.00),v40,z0,tPen\WObj:=wPaper;
    MoveL Offs(pOrigin,339.07,143.87,0.00),v40,fine,tPen\WObj:=wPaper;
    MoveL Offs(pOrigin,339.07,143.87,6.00),v60,z5,tPen\WObj:=wPaper;
    MoveL Offs(pOrigin,328.54,155.37,6.00),vTravel,z5,tPen\WObj:=wPaper;
    MoveL Offs(pOrigin,328.54,155.37,0.00),v60,z0,tPen\WObj:=wPaper;
    MoveL Offs(pOrigin,324.70,152.81,0.00),v40,z0,tPen\WObj:=wPaper;
    MoveL Offs(pOrigin,320.87,151.54,0.00),v40,z0,tPen\WObj:=wPaper;
    MoveL Offs(pOrigin,317.52,151.54,0.00),v40,z0,tPen\WObj:=wPaper;
    MoveL Offs(pOrigin,315.13,152.65,0.00),v40,z0,tPen\WObj:=wPaper;
    MoveL Offs(pOrigin,313.85,154.09,0.00),v40,z0,tPen\WObj:=wPaper;
    MoveL Offs(pOrigin,313.21,155.85,0.00),v40,z0,tPen\WObj:=wPaper;
    MoveL Offs(pOrigin,313.21,158.24,0.00),v40,z0,tPen\WObj:=wPaper;
    MoveL Offs(pOrigin,314.49,160.63,0.00),v40,z0,tPen\WObj:=wPaper;
    MoveL Offs(pOrigin,316.08,162.55,0.00),v40,z0,tPen\WObj:=wPaper;
    MoveL Offs(pOrigin,320.87,165.26,0.00),v40,z0,tPen\WObj:=wPaper;
    MoveL Offs(pOrigin,331.89,168.77,0.00),v40,z0,tPen\WObj:=wPaper;
    MoveL Offs(pOrigin,332.69,168.62,0.00),v40,z0,tPen\WObj:=wPaper;
    MoveL Offs(pOrigin,332.85,164.46,0.00),v40,z0,tPen\WObj:=wPaper;
    MoveL Offs(pOrigin,331.89,161.11,0.00),v40,z0,tPen\WObj:=wPaper;
    MoveL Offs(pOrigin,330.29,157.76,0.00),v40,z0,tPen\WObj:=wPaper;
    MoveL Offs(pOrigin,328.54,155.37,0.00),v40,fine,tPen\WObj:=wPaper;
    MoveL Offs(pOrigin,328.54,155.37,6.00),v60,z5,tPen\WObj:=wPaper;
    MoveL Offs(pOrigin,329.01,156.80,6.00),vTravel,z5,tPen\WObj:=wPaper;
    MoveL Offs(pOrigin,329.01,156.80,0.00),v60,z0,tPen\WObj:=wPaper;
    MoveL Offs(pOrigin,329.97,157.76,0.00),v40,z0,tPen\WObj:=wPaper;
    MoveL Offs(pOrigin,329.01,156.80,0.00),v40,fine,tPen\WObj:=wPaper;
    MoveL Offs(pOrigin,329.01,156.80,6.00),v60,z5,tPen\WObj:=wPaper;
    MoveL Offs(pOrigin,326.14,153.93,6.00),vTravel,z5,tPen\WObj:=wPaper;
    MoveL Offs(pOrigin,326.14,153.93,0.00),v60,z0,tPen\WObj:=wPaper;
    MoveL Offs(pOrigin,327.10,154.89,0.00),v40,z0,tPen\WObj:=wPaper;
    MoveL Offs(pOrigin,326.14,153.93,0.00),v40,fine,tPen\WObj:=wPaper;
    MoveL Offs(pOrigin,326.14,153.93,6.00),v60,z5,tPen\WObj:=wPaper;
    MoveL Offs(pOrigin,316.08,152.49,6.00),vTravel,z5,tPen\WObj:=wPaper;
    MoveL Offs(pOrigin,316.08,152.49,0.00),v60,z0,tPen\WObj:=wPaper;
    MoveL Offs(pOrigin,315.13,152.97,0.00),v40,z0,tPen\WObj:=wPaper;
    MoveL Offs(pOrigin,315.61,152.49,0.00),v40,z0,tPen\WObj:=wPaper;
    MoveL Offs(pOrigin,316.08,152.49,0.00),v40,z0,tPen\WObj:=wPaper;
    MoveL Offs(pOrigin,315.13,152.97,0.00),v40,z0,tPen\WObj:=wPaper;
    MoveL Offs(pOrigin,315.61,152.49,0.00),v40,z0,tPen\WObj:=wPaper;
    MoveL Offs(pOrigin,316.08,152.49,0.00),v40,fine,tPen\WObj:=wPaper;
    MoveL Offs(pOrigin,316.08,152.49,6.00),v60,z5,tPen\WObj:=wPaper;
    MoveL Offs(pOrigin,314.65,160.15,6.00),vTravel,z5,tPen\WObj:=wPaper;
    MoveL Offs(pOrigin,314.65,160.15,0.00),v60,z0,tPen\WObj:=wPaper;
    MoveL Offs(pOrigin,314.65,160.63,0.00),v40,z0,tPen\WObj:=wPaper;
    MoveL Offs(pOrigin,316.56,162.55,0.00),v40,z0,tPen\WObj:=wPaper;
    MoveL Offs(pOrigin,314.65,160.15,0.00),v40,z0,tPen\WObj:=wPaper;
    MoveL Offs(pOrigin,314.65,160.63,0.00),v40,z0,tPen\WObj:=wPaper;
    MoveL Offs(pOrigin,316.56,162.55,0.00),v40,z0,tPen\WObj:=wPaper;
    MoveL Offs(pOrigin,314.65,160.15,0.00),v40,fine,tPen\WObj:=wPaper;
    MoveL Offs(pOrigin,314.65,160.15,6.00),v60,z5,tPen\WObj:=wPaper;
    MoveL Offs(pOrigin,307.94,168.77,6.00),vTravel,z5,tPen\WObj:=wPaper;
    MoveL Offs(pOrigin,307.94,168.77,0.00),v60,z0,tPen\WObj:=wPaper;
    MoveL Offs(pOrigin,306.03,167.34,0.00),v40,z0,tPen\WObj:=wPaper;
    MoveL Offs(pOrigin,302.68,163.99,0.00),v40,z0,tPen\WObj:=wPaper;
    MoveL Offs(pOrigin,299.48,158.72,0.00),v40,z0,tPen\WObj:=wPaper;
    MoveL Offs(pOrigin,298.37,154.41,0.00),v40,z0,tPen\WObj:=wPaper;
    MoveL Offs(pOrigin,298.37,152.97,0.00),v40,z0,tPen\WObj:=wPaper;
    MoveL Offs(pOrigin,299.48,149.14,0.00),v40,z0,tPen\WObj:=wPaper;
    MoveL Offs(pOrigin,302.36,144.83,0.00),v40,z0,tPen\WObj:=wPaper;
    MoveL Offs(pOrigin,304.59,142.92,0.00),v40,z0,tPen\WObj:=wPaper;
    MoveL Offs(pOrigin,304.59,142.60,0.00),v40,z0,tPen\WObj:=wPaper;
    MoveL Offs(pOrigin,303.63,143.39,0.00),v40,z0,tPen\WObj:=wPaper;
    MoveL Offs(pOrigin,313.37,174.36,0.00),v40,z0,tPen\WObj:=wPaper;
    MoveL Offs(pOrigin,318.64,189.37,0.00),v40,z0,tPen\WObj:=wPaper;
    MoveL Offs(pOrigin,322.31,184.58,0.00),v40,z0,tPen\WObj:=wPaper;
    MoveL Offs(pOrigin,327.58,179.31,0.00),v40,z0,tPen\WObj:=wPaper;
    MoveL Offs(pOrigin,328.06,178.35,0.00),v40,z0,tPen\WObj:=wPaper;
    MoveL Offs(pOrigin,328.06,177.39,0.00),v40,z0,tPen\WObj:=wPaper;
    MoveL Offs(pOrigin,327.58,176.92,0.00),v40,z0,tPen\WObj:=wPaper;
    MoveL Offs(pOrigin,325.18,176.44,0.00),v40,z0,tPen\WObj:=wPaper;
    MoveL Offs(pOrigin,314.65,172.77,0.00),v40,z0,tPen\WObj:=wPaper;
    MoveL Offs(pOrigin,307.94,168.77,0.00),v40,z0,tPen\WObj:=wPaper;
    MoveL Offs(pOrigin,306.99,168.30,0.00),v40,z0,tPen\WObj:=wPaper;
    MoveL Offs(pOrigin,307.94,169.25,0.00),v40,z0,tPen\WObj:=wPaper;
    MoveL Offs(pOrigin,306.99,168.30,0.00),v40,fine,tPen\WObj:=wPaper;
    MoveL Offs(pOrigin,306.99,168.30,6.00),v60,z5,tPen\WObj:=wPaper;
    MoveL Offs(pOrigin,303.63,165.42,6.00),vTravel,z5,tPen\WObj:=wPaper;
    MoveL Offs(pOrigin,303.63,165.42,0.00),v60,z0,tPen\WObj:=wPaper;
    MoveL Offs(pOrigin,306.03,167.82,0.00),v40,z0,tPen\WObj:=wPaper;
    MoveL Offs(pOrigin,303.63,165.42,0.00),v40,fine,tPen\WObj:=wPaper;
    MoveL Offs(pOrigin,303.63,165.42,6.00),v60,z5,tPen\WObj:=wPaper;
    MoveL Offs(pOrigin,302.20,163.99,6.00),vTravel,z5,tPen\WObj:=wPaper;
    MoveL Offs(pOrigin,302.20,163.99,0.00),v60,z0,tPen\WObj:=wPaper;
    MoveL Offs(pOrigin,303.15,164.94,0.00),v40,z0,tPen\WObj:=wPaper;
    MoveL Offs(pOrigin,302.20,163.99,0.00),v40,fine,tPen\WObj:=wPaper;
    MoveL Offs(pOrigin,302.20,163.99,6.00),v60,z5,tPen\WObj:=wPaper;
    MoveL Offs(pOrigin,298.37,175.00,6.00),vTravel,z5,tPen\WObj:=wPaper;
    MoveL Offs(pOrigin,298.37,175.00,0.00),v60,z0,tPen\WObj:=wPaper;
    MoveL Offs(pOrigin,299.80,176.44,0.00),v40,z0,tPen\WObj:=wPaper;
    MoveL Offs(pOrigin,297.89,175.00,0.00),v40,z0,tPen\WObj:=wPaper;
    MoveL Offs(pOrigin,298.37,175.00,0.00),v40,z0,tPen\WObj:=wPaper;
    MoveL Offs(pOrigin,299.80,176.44,0.00),v40,z0,tPen\WObj:=wPaper;
    MoveL Offs(pOrigin,297.89,175.00,0.00),v40,z0,tPen\WObj:=wPaper;
    MoveL Offs(pOrigin,298.37,175.00,0.00),v40,fine,tPen\WObj:=wPaper;
    MoveL Offs(pOrigin,298.37,175.00,6.00),v60,z5,tPen\WObj:=wPaper;
    MoveL Offs(pOrigin,301.24,177.39,6.00),vTravel,z5,tPen\WObj:=wPaper;
    MoveL Offs(pOrigin,301.24,177.39,0.00),v60,z0,tPen\WObj:=wPaper;
    MoveL Offs(pOrigin,302.20,178.35,0.00),v40,z0,tPen\WObj:=wPaper;
    MoveL Offs(pOrigin,301.24,177.39,0.00),v40,fine,tPen\WObj:=wPaper;
    MoveL Offs(pOrigin,301.24,177.39,6.00),v60,z5,tPen\WObj:=wPaper;
    MoveL Offs(pOrigin,303.15,179.79,6.00),vTravel,z5,tPen\WObj:=wPaper;
    MoveL Offs(pOrigin,303.15,179.79,0.00),v60,z0,tPen\WObj:=wPaper;
    MoveL Offs(pOrigin,303.63,180.27,0.00),v40,z0,tPen\WObj:=wPaper;
    MoveL Offs(pOrigin,303.63,180.75,0.00),v40,z0,tPen\WObj:=wPaper;
    MoveL Offs(pOrigin,303.15,179.79,0.00),v40,z0,tPen\WObj:=wPaper;
    MoveL Offs(pOrigin,303.63,180.27,0.00),v40,z0,tPen\WObj:=wPaper;
    MoveL Offs(pOrigin,303.63,180.75,0.00),v40,z0,tPen\WObj:=wPaper;
    MoveL Offs(pOrigin,303.15,179.79,0.00),v40,fine,tPen\WObj:=wPaper;
    MoveL Offs(pOrigin,303.15,179.79,6.00),v60,z5,tPen\WObj:=wPaper;
    MoveL Offs(pOrigin,299.32,186.01,6.00),vTravel,z5,tPen\WObj:=wPaper;
    MoveL Offs(pOrigin,299.32,186.01,0.00),v60,z0,tPen\WObj:=wPaper;
    MoveL Offs(pOrigin,299.32,186.49,0.00),v40,z0,tPen\WObj:=wPaper;
    MoveL Offs(pOrigin,299.80,186.49,0.00),v40,z0,tPen\WObj:=wPaper;
    MoveL Offs(pOrigin,300.28,186.97,0.00),v40,z0,tPen\WObj:=wPaper;
  ENDPROC

  PROC DrawPart31()
    MoveL Offs(pOrigin,299.32,186.01,0.00),v40,z0,tPen\WObj:=wPaper;
    MoveL Offs(pOrigin,299.32,186.49,0.00),v40,z0,tPen\WObj:=wPaper;
    MoveL Offs(pOrigin,299.80,186.49,0.00),v40,z0,tPen\WObj:=wPaper;
    MoveL Offs(pOrigin,300.28,186.97,0.00),v40,z0,tPen\WObj:=wPaper;
    MoveL Offs(pOrigin,299.32,186.01,0.00),v40,fine,tPen\WObj:=wPaper;
    MoveL Offs(pOrigin,299.32,186.01,6.00),v60,z5,tPen\WObj:=wPaper;
    MoveL Offs(pOrigin,297.41,184.58,6.00),vTravel,z5,tPen\WObj:=wPaper;
    MoveL Offs(pOrigin,297.41,184.58,0.00),v60,z0,tPen\WObj:=wPaper;
    MoveL Offs(pOrigin,296.45,183.62,0.00),v40,z0,tPen\WObj:=wPaper;
    MoveL Offs(pOrigin,296.45,184.10,0.00),v40,z0,tPen\WObj:=wPaper;
    MoveL Offs(pOrigin,296.93,184.10,0.00),v40,z0,tPen\WObj:=wPaper;
    MoveL Offs(pOrigin,297.41,184.58,0.00),v40,z0,tPen\WObj:=wPaper;
    MoveL Offs(pOrigin,296.45,183.62,0.00),v40,z0,tPen\WObj:=wPaper;
    MoveL Offs(pOrigin,296.45,184.10,0.00),v40,z0,tPen\WObj:=wPaper;
    MoveL Offs(pOrigin,296.93,184.10,0.00),v40,z0,tPen\WObj:=wPaper;
    MoveL Offs(pOrigin,297.41,184.58,0.00),v40,fine,tPen\WObj:=wPaper;
    MoveL Offs(pOrigin,297.41,184.58,6.00),v60,z5,tPen\WObj:=wPaper;
    MoveL Offs(pOrigin,295.49,183.14,6.00),vTravel,z5,tPen\WObj:=wPaper;
    MoveL Offs(pOrigin,295.49,183.14,0.00),v60,z0,tPen\WObj:=wPaper;
    MoveL Offs(pOrigin,295.01,182.66,0.00),v40,z0,tPen\WObj:=wPaper;
    MoveL Offs(pOrigin,295.01,183.14,0.00),v40,z0,tPen\WObj:=wPaper;
    MoveL Offs(pOrigin,295.49,183.14,0.00),v40,z0,tPen\WObj:=wPaper;
    MoveL Offs(pOrigin,295.01,182.66,0.00),v40,z0,tPen\WObj:=wPaper;
    MoveL Offs(pOrigin,295.01,183.14,0.00),v40,z0,tPen\WObj:=wPaper;
    MoveL Offs(pOrigin,295.49,183.14,0.00),v40,fine,tPen\WObj:=wPaper;
    MoveL Offs(pOrigin,295.49,183.14,6.00),v60,z5,tPen\WObj:=wPaper;
    MoveL Offs(pOrigin,285.92,192.72,6.00),vTravel,z5,tPen\WObj:=wPaper;
    MoveL Offs(pOrigin,285.92,192.72,0.00),v60,z0,tPen\WObj:=wPaper;
    MoveL Offs(pOrigin,285.92,193.20,0.00),v40,z0,tPen\WObj:=wPaper;
    MoveL Offs(pOrigin,285.44,193.68,0.00),v40,z0,tPen\WObj:=wPaper;
    MoveL Offs(pOrigin,285.92,192.72,0.00),v40,z0,tPen\WObj:=wPaper;
    MoveL Offs(pOrigin,285.92,193.20,0.00),v40,z0,tPen\WObj:=wPaper;
    MoveL Offs(pOrigin,285.44,193.68,0.00),v40,z0,tPen\WObj:=wPaper;
    MoveL Offs(pOrigin,285.92,192.72,0.00),v40,fine,tPen\WObj:=wPaper;
    MoveL Offs(pOrigin,285.92,192.72,6.00),v60,z5,tPen\WObj:=wPaper;
    MoveL Offs(pOrigin,284.48,195.11,6.00),vTravel,z5,tPen\WObj:=wPaper;
    MoveL Offs(pOrigin,284.48,195.11,0.00),v60,z0,tPen\WObj:=wPaper;
    MoveL Offs(pOrigin,284.48,195.59,0.00),v40,z0,tPen\WObj:=wPaper;
    MoveL Offs(pOrigin,284.00,196.07,0.00),v40,z0,tPen\WObj:=wPaper;
    MoveL Offs(pOrigin,284.48,195.11,0.00),v40,z0,tPen\WObj:=wPaper;
    MoveL Offs(pOrigin,284.48,195.59,0.00),v40,z0,tPen\WObj:=wPaper;
    MoveL Offs(pOrigin,284.00,196.07,0.00),v40,z0,tPen\WObj:=wPaper;
    MoveL Offs(pOrigin,284.48,195.11,0.00),v40,fine,tPen\WObj:=wPaper;
    MoveL Offs(pOrigin,284.48,195.11,6.00),v60,z5,tPen\WObj:=wPaper;
    MoveL Offs(pOrigin,283.04,197.03,6.00),vTravel,z5,tPen\WObj:=wPaper;
    MoveL Offs(pOrigin,283.04,197.03,0.00),v60,z0,tPen\WObj:=wPaper;
    MoveL Offs(pOrigin,283.04,197.51,0.00),v40,z0,tPen\WObj:=wPaper;
    MoveL Offs(pOrigin,282.56,197.51,0.00),v40,z0,tPen\WObj:=wPaper;
    MoveL Offs(pOrigin,281.61,198.46,0.00),v40,z0,tPen\WObj:=wPaper;
    MoveL Offs(pOrigin,283.04,197.03,0.00),v40,z0,tPen\WObj:=wPaper;
    MoveL Offs(pOrigin,283.04,197.51,0.00),v40,z0,tPen\WObj:=wPaper;
    MoveL Offs(pOrigin,282.56,197.51,0.00),v40,z0,tPen\WObj:=wPaper;
    MoveL Offs(pOrigin,281.61,198.46,0.00),v40,z0,tPen\WObj:=wPaper;
    MoveL Offs(pOrigin,283.04,197.03,0.00),v40,fine,tPen\WObj:=wPaper;
    MoveL Offs(pOrigin,283.04,197.03,6.00),v60,z5,tPen\WObj:=wPaper;
    MoveL Offs(pOrigin,281.13,198.94,6.00),vTravel,z5,tPen\WObj:=wPaper;
    MoveL Offs(pOrigin,281.13,198.94,0.00),v60,z0,tPen\WObj:=wPaper;
    MoveL Offs(pOrigin,281.13,199.42,0.00),v40,z0,tPen\WObj:=wPaper;
    MoveL Offs(pOrigin,280.65,199.42,0.00),v40,z0,tPen\WObj:=wPaper;
    MoveL Offs(pOrigin,279.21,200.86,0.00),v40,z0,tPen\WObj:=wPaper;
    MoveL Offs(pOrigin,281.13,198.94,0.00),v40,z0,tPen\WObj:=wPaper;
    MoveL Offs(pOrigin,281.13,199.42,0.00),v40,z0,tPen\WObj:=wPaper;
    MoveL Offs(pOrigin,280.65,199.42,0.00),v40,z0,tPen\WObj:=wPaper;
    MoveL Offs(pOrigin,279.21,200.86,0.00),v40,z0,tPen\WObj:=wPaper;
    MoveL Offs(pOrigin,281.13,198.94,0.00),v40,fine,tPen\WObj:=wPaper;
    MoveL Offs(pOrigin,281.13,198.94,6.00),v60,z5,tPen\WObj:=wPaper;
    MoveL Offs(pOrigin,297.41,198.46,6.00),vTravel,z5,tPen\WObj:=wPaper;
    MoveL Offs(pOrigin,297.41,198.46,0.00),v60,z0,tPen\WObj:=wPaper;
    MoveL Offs(pOrigin,297.41,200.38,0.00),v40,z0,tPen\WObj:=wPaper;
    MoveL Offs(pOrigin,297.41,198.46,0.00),v40,z0,tPen\WObj:=wPaper;
    MoveL Offs(pOrigin,298.37,198.46,0.00),v40,z0,tPen\WObj:=wPaper;
    MoveL Offs(pOrigin,299.32,198.46,0.00),v40,z0,tPen\WObj:=wPaper;
    MoveL Offs(pOrigin,300.28,199.42,0.00),v40,z0,tPen\WObj:=wPaper;
    MoveL Offs(pOrigin,300.76,199.42,0.00),v40,z0,tPen\WObj:=wPaper;
    MoveL Offs(pOrigin,300.28,198.94,0.00),v40,z0,tPen\WObj:=wPaper;
    MoveL Offs(pOrigin,298.37,198.46,0.00),v40,z0,tPen\WObj:=wPaper;
    MoveL Offs(pOrigin,299.32,198.46,0.00),v40,z0,tPen\WObj:=wPaper;
    MoveL Offs(pOrigin,300.28,199.42,0.00),v40,z0,tPen\WObj:=wPaper;
    MoveL Offs(pOrigin,300.76,199.42,0.00),v40,z0,tPen\WObj:=wPaper;
    MoveL Offs(pOrigin,300.28,198.94,0.00),v40,z0,tPen\WObj:=wPaper;
    MoveL Offs(pOrigin,298.37,198.46,0.00),v40,fine,tPen\WObj:=wPaper;
    MoveL Offs(pOrigin,298.37,198.46,6.00),v60,z5,tPen\WObj:=wPaper;
    MoveL Offs(pOrigin,297.89,200.38,6.00),vTravel,z5,tPen\WObj:=wPaper;
    MoveL Offs(pOrigin,297.89,200.38,0.00),v60,z0,tPen\WObj:=wPaper;
    MoveL Offs(pOrigin,297.89,200.86,0.00),v40,z0,tPen\WObj:=wPaper;
    MoveL Offs(pOrigin,298.85,201.82,0.00),v40,z0,tPen\WObj:=wPaper;
    MoveL Offs(pOrigin,297.89,200.38,0.00),v40,z0,tPen\WObj:=wPaper;
    MoveL Offs(pOrigin,297.89,200.86,0.00),v40,z0,tPen\WObj:=wPaper;
    MoveL Offs(pOrigin,298.85,201.82,0.00),v40,z0,tPen\WObj:=wPaper;
    MoveL Offs(pOrigin,297.89,200.38,0.00),v40,z0,tPen\WObj:=wPaper;
    MoveL Offs(pOrigin,297.89,201.34,0.00),v40,z0,tPen\WObj:=wPaper;
    MoveL Offs(pOrigin,298.85,202.30,0.00),v40,z0,tPen\WObj:=wPaper;
    MoveL Offs(pOrigin,298.85,202.77,0.00),v40,z0,tPen\WObj:=wPaper;
    MoveL Offs(pOrigin,299.32,203.25,0.00),v40,z0,tPen\WObj:=wPaper;
    MoveL Offs(pOrigin,299.80,203.25,0.00),v40,z0,tPen\WObj:=wPaper;
    MoveL Offs(pOrigin,297.89,201.34,0.00),v40,z0,tPen\WObj:=wPaper;
    MoveL Offs(pOrigin,298.85,202.30,0.00),v40,z0,tPen\WObj:=wPaper;
    MoveL Offs(pOrigin,298.85,202.77,0.00),v40,z0,tPen\WObj:=wPaper;
    MoveL Offs(pOrigin,299.32,203.25,0.00),v40,z0,tPen\WObj:=wPaper;
    MoveL Offs(pOrigin,299.80,203.25,0.00),v40,z0,tPen\WObj:=wPaper;
    MoveL Offs(pOrigin,297.89,201.34,0.00),v40,fine,tPen\WObj:=wPaper;
    MoveL Offs(pOrigin,297.89,201.34,6.00),v60,z5,tPen\WObj:=wPaper;
    MoveL Offs(pOrigin,299.80,203.73,6.00),vTravel,z5,tPen\WObj:=wPaper;
    MoveL Offs(pOrigin,299.80,203.73,0.00),v60,z0,tPen\WObj:=wPaper;
    MoveL Offs(pOrigin,300.28,205.17,0.00),v40,z0,tPen\WObj:=wPaper;
    MoveL Offs(pOrigin,301.72,206.61,0.00),v40,z0,tPen\WObj:=wPaper;
    MoveL Offs(pOrigin,299.80,203.73,0.00),v40,z0,tPen\WObj:=wPaper;
    MoveL Offs(pOrigin,300.28,205.17,0.00),v40,z0,tPen\WObj:=wPaper;
    MoveL Offs(pOrigin,301.72,206.61,0.00),v40,z0,tPen\WObj:=wPaper;
    MoveL Offs(pOrigin,299.80,203.73,0.00),v40,z0,tPen\WObj:=wPaper;
    MoveL Offs(pOrigin,300.28,204.21,0.00),v40,z0,tPen\WObj:=wPaper;
    MoveL Offs(pOrigin,300.28,204.69,0.00),v40,z0,tPen\WObj:=wPaper;
    MoveL Offs(pOrigin,300.76,205.17,0.00),v40,z0,tPen\WObj:=wPaper;
    MoveL Offs(pOrigin,300.28,204.21,0.00),v40,z0,tPen\WObj:=wPaper;
    MoveL Offs(pOrigin,300.28,204.69,0.00),v40,z0,tPen\WObj:=wPaper;
    MoveL Offs(pOrigin,300.76,205.17,0.00),v40,z0,tPen\WObj:=wPaper;
    MoveL Offs(pOrigin,300.28,204.21,0.00),v40,fine,tPen\WObj:=wPaper;
    MoveL Offs(pOrigin,300.28,204.21,6.00),v60,z5,tPen\WObj:=wPaper;
    MoveL Offs(pOrigin,301.24,206.61,6.00),vTravel,z5,tPen\WObj:=wPaper;
    MoveL Offs(pOrigin,301.24,206.61,0.00),v60,z0,tPen\WObj:=wPaper;
  ENDPROC

  PROC DrawPart32()
    MoveL Offs(pOrigin,302.52,208.52,0.00),v40,z0,tPen\WObj:=wPaper;
    MoveL Offs(pOrigin,302.68,209.48,0.00),v40,z0,tPen\WObj:=wPaper;
    MoveL Offs(pOrigin,301.08,211.39,0.00),v40,z0,tPen\WObj:=wPaper;
    MoveL Offs(pOrigin,300.28,213.79,0.00),v40,z0,tPen\WObj:=wPaper;
    MoveL Offs(pOrigin,300.28,215.70,0.00),v40,z0,tPen\WObj:=wPaper;
    MoveL Offs(pOrigin,301.24,206.61,0.00),v40,fine,tPen\WObj:=wPaper;
    MoveL Offs(pOrigin,301.24,206.61,6.00),v60,z5,tPen\WObj:=wPaper;
    MoveL Offs(pOrigin,302.20,209.96,6.00),vTravel,z5,tPen\WObj:=wPaper;
    MoveL Offs(pOrigin,302.20,209.96,0.00),v60,z0,tPen\WObj:=wPaper;
    MoveL Offs(pOrigin,301.72,210.92,0.00),v40,z0,tPen\WObj:=wPaper;
    MoveL Offs(pOrigin,302.20,210.44,0.00),v40,z0,tPen\WObj:=wPaper;
    MoveL Offs(pOrigin,302.20,209.96,0.00),v40,z0,tPen\WObj:=wPaper;
    MoveL Offs(pOrigin,301.72,210.92,0.00),v40,z0,tPen\WObj:=wPaper;
    MoveL Offs(pOrigin,302.20,210.44,0.00),v40,z0,tPen\WObj:=wPaper;
    MoveL Offs(pOrigin,302.20,209.96,0.00),v40,fine,tPen\WObj:=wPaper;
    MoveL Offs(pOrigin,302.20,209.96,6.00),v60,z5,tPen\WObj:=wPaper;
    MoveL Offs(pOrigin,300.28,216.66,6.00),vTravel,z5,tPen\WObj:=wPaper;
    MoveL Offs(pOrigin,300.28,216.66,0.00),v60,z0,tPen\WObj:=wPaper;
    MoveL Offs(pOrigin,300.28,218.58,0.00),v40,z0,tPen\WObj:=wPaper;
    MoveL Offs(pOrigin,300.76,219.06,0.00),v40,z0,tPen\WObj:=wPaper;
    MoveL Offs(pOrigin,300.76,220.49,0.00),v40,z0,tPen\WObj:=wPaper;
    MoveL Offs(pOrigin,300.28,216.66,0.00),v40,z0,tPen\WObj:=wPaper;
    MoveL Offs(pOrigin,300.28,218.58,0.00),v40,z0,tPen\WObj:=wPaper;
    MoveL Offs(pOrigin,300.76,219.06,0.00),v40,z0,tPen\WObj:=wPaper;
    MoveL Offs(pOrigin,300.76,220.49,0.00),v40,z0,tPen\WObj:=wPaper;
    MoveL Offs(pOrigin,300.28,216.66,0.00),v40,fine,tPen\WObj:=wPaper;
    MoveL Offs(pOrigin,300.28,216.66,6.00),v60,z5,tPen\WObj:=wPaper;
    MoveL Offs(pOrigin,301.24,221.45,6.00),vTravel,z5,tPen\WObj:=wPaper;
    MoveL Offs(pOrigin,301.24,221.45,0.00),v60,z0,tPen\WObj:=wPaper;
    MoveL Offs(pOrigin,302.68,224.32,0.00),v40,z0,tPen\WObj:=wPaper;
    MoveL Offs(pOrigin,305.07,226.72,0.00),v40,z0,tPen\WObj:=wPaper;
    MoveL Offs(pOrigin,307.46,228.00,0.00),v40,z0,tPen\WObj:=wPaper;
    MoveL Offs(pOrigin,301.24,221.45,0.00),v40,fine,tPen\WObj:=wPaper;
    MoveL Offs(pOrigin,301.24,221.45,6.00),v60,z5,tPen\WObj:=wPaper;
    MoveL Offs(pOrigin,302.20,222.89,6.00),vTravel,z5,tPen\WObj:=wPaper;
    MoveL Offs(pOrigin,302.20,222.89,0.00),v60,z0,tPen\WObj:=wPaper;
    MoveL Offs(pOrigin,302.20,223.37,0.00),v40,z0,tPen\WObj:=wPaper;
    MoveL Offs(pOrigin,305.55,226.72,0.00),v40,z0,tPen\WObj:=wPaper;
    MoveL Offs(pOrigin,302.20,222.89,0.00),v40,z0,tPen\WObj:=wPaper;
    MoveL Offs(pOrigin,302.20,223.37,0.00),v40,z0,tPen\WObj:=wPaper;
    MoveL Offs(pOrigin,305.55,226.72,0.00),v40,z0,tPen\WObj:=wPaper;
    MoveL Offs(pOrigin,302.20,222.89,0.00),v40,fine,tPen\WObj:=wPaper;
    MoveL Offs(pOrigin,302.20,222.89,6.00),v60,z5,tPen\WObj:=wPaper;
    MoveL Offs(pOrigin,308.58,228.47,6.00),vTravel,z5,tPen\WObj:=wPaper;
    MoveL Offs(pOrigin,308.58,228.47,0.00),v60,z0,tPen\WObj:=wPaper;
    MoveL Offs(pOrigin,310.34,229.11,0.00),v40,z0,tPen\WObj:=wPaper;
    MoveL Offs(pOrigin,311.77,229.11,0.00),v40,z0,tPen\WObj:=wPaper;
    MoveL Offs(pOrigin,313.85,228.31,0.00),v40,z0,tPen\WObj:=wPaper;
    MoveL Offs(pOrigin,312.09,228.15,0.00),v40,z0,tPen\WObj:=wPaper;
    MoveL Offs(pOrigin,308.58,228.47,0.00),v40,fine,tPen\WObj:=wPaper;
    MoveL Offs(pOrigin,308.58,228.47,6.00),v60,z5,tPen\WObj:=wPaper;
    MoveL Offs(pOrigin,314.81,227.84,6.00),vTravel,z5,tPen\WObj:=wPaper;
    MoveL Offs(pOrigin,314.81,227.84,0.00),v60,z0,tPen\WObj:=wPaper;
    MoveL Offs(pOrigin,310.98,208.04,0.00),v40,z0,tPen\WObj:=wPaper;
    MoveL Offs(pOrigin,314.01,212.35,0.00),v40,z0,tPen\WObj:=wPaper;
    MoveL Offs(pOrigin,315.29,214.75,0.00),v40,z0,tPen\WObj:=wPaper;
    MoveL Offs(pOrigin,316.56,218.10,0.00),v40,z0,tPen\WObj:=wPaper;
    MoveL Offs(pOrigin,317.52,221.93,0.00),v40,z0,tPen\WObj:=wPaper;
    MoveL Offs(pOrigin,315.92,226.72,0.00),v40,z0,tPen\WObj:=wPaper;
    MoveL Offs(pOrigin,314.81,227.84,0.00),v40,fine,tPen\WObj:=wPaper;
    MoveL Offs(pOrigin,314.81,227.84,6.00),v60,z5,tPen\WObj:=wPaper;
    MoveL Offs(pOrigin,323.75,215.23,6.00),vTravel,z5,tPen\WObj:=wPaper;
    MoveL Offs(pOrigin,323.75,215.23,0.00),v60,z0,tPen\WObj:=wPaper;
    MoveL Offs(pOrigin,329.01,219.22,0.00),v40,z0,tPen\WObj:=wPaper;
    MoveL Offs(pOrigin,331.89,220.49,0.00),v40,z0,tPen\WObj:=wPaper;
    MoveL Offs(pOrigin,324.07,213.63,0.00),v40,z0,tPen\WObj:=wPaper;
    MoveL Offs(pOrigin,319.92,210.44,0.00),v40,z0,tPen\WObj:=wPaper;
    MoveL Offs(pOrigin,322.31,213.79,0.00),v40,z0,tPen\WObj:=wPaper;
    MoveL Offs(pOrigin,323.75,215.23,0.00),v40,z0,tPen\WObj:=wPaper;
    MoveL Offs(pOrigin,324.23,215.23,0.00),v40,z0,tPen\WObj:=wPaper;
    MoveL Offs(pOrigin,322.79,213.79,0.00),v40,z0,tPen\WObj:=wPaper;
    MoveL Offs(pOrigin,322.79,214.27,0.00),v40,z0,tPen\WObj:=wPaper;
    MoveL Offs(pOrigin,323.27,214.27,0.00),v40,z0,tPen\WObj:=wPaper;
    MoveL Offs(pOrigin,324.23,215.23,0.00),v40,z0,tPen\WObj:=wPaper;
    MoveL Offs(pOrigin,322.79,213.79,0.00),v40,z0,tPen\WObj:=wPaper;
    MoveL Offs(pOrigin,322.79,214.27,0.00),v40,z0,tPen\WObj:=wPaper;
    MoveL Offs(pOrigin,323.27,214.27,0.00),v40,z0,tPen\WObj:=wPaper;
    MoveL Offs(pOrigin,324.23,215.23,0.00),v40,z0,tPen\WObj:=wPaper;
    MoveL Offs(pOrigin,325.18,215.70,0.00),v40,z0,tPen\WObj:=wPaper;
    MoveL Offs(pOrigin,325.18,216.18,0.00),v40,z0,tPen\WObj:=wPaper;
    MoveL Offs(pOrigin,325.66,216.18,0.00),v40,z0,tPen\WObj:=wPaper;
    MoveL Offs(pOrigin,326.62,217.14,0.00),v40,z0,tPen\WObj:=wPaper;
    MoveL Offs(pOrigin,325.18,215.70,0.00),v40,z0,tPen\WObj:=wPaper;
    MoveL Offs(pOrigin,325.18,216.18,0.00),v40,z0,tPen\WObj:=wPaper;
    MoveL Offs(pOrigin,325.66,216.18,0.00),v40,z0,tPen\WObj:=wPaper;
    MoveL Offs(pOrigin,326.62,217.14,0.00),v40,z0,tPen\WObj:=wPaper;
    MoveL Offs(pOrigin,325.18,215.70,0.00),v40,fine,tPen\WObj:=wPaper;
    MoveL Offs(pOrigin,325.18,215.70,6.00),v60,z5,tPen\WObj:=wPaper;
    MoveL Offs(pOrigin,328.06,218.10,6.00),vTravel,z5,tPen\WObj:=wPaper;
    MoveL Offs(pOrigin,328.06,218.10,0.00),v60,z0,tPen\WObj:=wPaper;
    MoveL Offs(pOrigin,328.06,218.58,0.00),v40,z0,tPen\WObj:=wPaper;
    MoveL Offs(pOrigin,328.54,218.58,0.00),v40,z0,tPen\WObj:=wPaper;
    MoveL Offs(pOrigin,328.06,218.10,0.00),v40,z0,tPen\WObj:=wPaper;
    MoveL Offs(pOrigin,328.06,218.58,0.00),v40,z0,tPen\WObj:=wPaper;
    MoveL Offs(pOrigin,328.54,218.58,0.00),v40,z0,tPen\WObj:=wPaper;
    MoveL Offs(pOrigin,328.06,218.10,0.00),v40,fine,tPen\WObj:=wPaper;
    MoveL Offs(pOrigin,328.06,218.10,6.00),v60,z5,tPen\WObj:=wPaper;
    MoveL Offs(pOrigin,321.83,212.35,6.00),vTravel,z5,tPen\WObj:=wPaper;
    MoveL Offs(pOrigin,321.83,212.35,0.00),v60,z0,tPen\WObj:=wPaper;
    MoveL Offs(pOrigin,320.87,211.39,0.00),v40,z0,tPen\WObj:=wPaper;
    MoveL Offs(pOrigin,320.87,211.87,0.00),v40,z0,tPen\WObj:=wPaper;
    MoveL Offs(pOrigin,321.35,211.87,0.00),v40,z0,tPen\WObj:=wPaper;
    MoveL Offs(pOrigin,321.83,212.35,0.00),v40,z0,tPen\WObj:=wPaper;
    MoveL Offs(pOrigin,320.87,211.39,0.00),v40,z0,tPen\WObj:=wPaper;
    MoveL Offs(pOrigin,320.87,211.87,0.00),v40,z0,tPen\WObj:=wPaper;
    MoveL Offs(pOrigin,321.35,211.87,0.00),v40,z0,tPen\WObj:=wPaper;
    MoveL Offs(pOrigin,321.83,212.35,0.00),v40,fine,tPen\WObj:=wPaper;
    MoveL Offs(pOrigin,321.83,212.35,6.00),v60,z5,tPen\WObj:=wPaper;
    MoveL Offs(pOrigin,319.92,209.48,6.00),vTravel,z5,tPen\WObj:=wPaper;
    MoveL Offs(pOrigin,319.92,209.48,0.00),v60,z0,tPen\WObj:=wPaper;
    MoveL Offs(pOrigin,318.00,206.61,0.00),v40,z0,tPen\WObj:=wPaper;
    MoveL Offs(pOrigin,318.00,207.08,0.00),v40,z0,tPen\WObj:=wPaper;
    MoveL Offs(pOrigin,318.96,208.04,0.00),v40,z0,tPen\WObj:=wPaper;
    MoveL Offs(pOrigin,318.96,209.00,0.00),v40,z0,tPen\WObj:=wPaper;
    MoveL Offs(pOrigin,319.44,209.48,0.00),v40,z0,tPen\WObj:=wPaper;
    MoveL Offs(pOrigin,319.92,209.48,0.00),v40,z0,tPen\WObj:=wPaper;
    MoveL Offs(pOrigin,318.00,206.61,0.00),v40,z0,tPen\WObj:=wPaper;
    MoveL Offs(pOrigin,318.00,207.08,0.00),v40,z0,tPen\WObj:=wPaper;
    MoveL Offs(pOrigin,318.96,208.04,0.00),v40,z0,tPen\WObj:=wPaper;
    MoveL Offs(pOrigin,318.96,209.00,0.00),v40,z0,tPen\WObj:=wPaper;
  ENDPROC

  PROC DrawPart33()
    MoveL Offs(pOrigin,319.44,209.48,0.00),v40,z0,tPen\WObj:=wPaper;
    MoveL Offs(pOrigin,319.92,209.48,0.00),v40,fine,tPen\WObj:=wPaper;
    MoveL Offs(pOrigin,319.92,209.48,6.00),v60,z5,tPen\WObj:=wPaper;
    MoveL Offs(pOrigin,317.68,205.97,6.00),vTravel,z5,tPen\WObj:=wPaper;
    MoveL Offs(pOrigin,317.68,205.97,0.00),v60,z0,tPen\WObj:=wPaper;
    MoveL Offs(pOrigin,316.56,194.15,0.00),v40,z0,tPen\WObj:=wPaper;
    MoveL Offs(pOrigin,316.08,195.59,0.00),v40,z0,tPen\WObj:=wPaper;
    MoveL Offs(pOrigin,316.08,199.90,0.00),v40,z0,tPen\WObj:=wPaper;
    MoveL Offs(pOrigin,317.68,205.97,0.00),v40,fine,tPen\WObj:=wPaper;
    MoveL Offs(pOrigin,317.68,205.97,6.00),v60,z5,tPen\WObj:=wPaper;
    MoveL Offs(pOrigin,312.73,209.96,6.00),vTravel,z5,tPen\WObj:=wPaper;
    MoveL Offs(pOrigin,312.73,209.96,0.00),v60,z0,tPen\WObj:=wPaper;
    MoveL Offs(pOrigin,311.77,208.52,0.00),v40,z0,tPen\WObj:=wPaper;
    MoveL Offs(pOrigin,311.77,209.00,0.00),v40,z0,tPen\WObj:=wPaper;
    MoveL Offs(pOrigin,312.73,209.96,0.00),v40,z0,tPen\WObj:=wPaper;
    MoveL Offs(pOrigin,311.77,208.52,0.00),v40,z0,tPen\WObj:=wPaper;
    MoveL Offs(pOrigin,311.77,209.00,0.00),v40,z0,tPen\WObj:=wPaper;
    MoveL Offs(pOrigin,312.73,209.96,0.00),v40,fine,tPen\WObj:=wPaper;
    MoveL Offs(pOrigin,312.73,209.96,6.00),v60,z5,tPen\WObj:=wPaper;
    MoveL Offs(pOrigin,313.69,211.39,6.00),vTravel,z5,tPen\WObj:=wPaper;
    MoveL Offs(pOrigin,313.69,211.39,0.00),v60,z0,tPen\WObj:=wPaper;
    MoveL Offs(pOrigin,313.69,211.87,0.00),v40,z0,tPen\WObj:=wPaper;
    MoveL Offs(pOrigin,314.17,211.87,0.00),v40,z0,tPen\WObj:=wPaper;
    MoveL Offs(pOrigin,313.69,211.39,0.00),v40,z0,tPen\WObj:=wPaper;
    MoveL Offs(pOrigin,313.69,211.87,0.00),v40,z0,tPen\WObj:=wPaper;
    MoveL Offs(pOrigin,314.17,211.87,0.00),v40,z0,tPen\WObj:=wPaper;
    MoveL Offs(pOrigin,313.69,211.39,0.00),v40,fine,tPen\WObj:=wPaper;
    MoveL Offs(pOrigin,313.69,211.39,6.00),v60,z5,tPen\WObj:=wPaper;
    MoveL Offs(pOrigin,310.34,207.56,6.00),vTravel,z5,tPen\WObj:=wPaper;
    MoveL Offs(pOrigin,310.34,207.56,0.00),v60,z0,tPen\WObj:=wPaper;
    MoveL Offs(pOrigin,308.42,204.69,0.00),v40,z0,tPen\WObj:=wPaper;
    MoveL Offs(pOrigin,308.42,205.17,0.00),v40,z0,tPen\WObj:=wPaper;
    MoveL Offs(pOrigin,310.34,207.08,0.00),v40,z0,tPen\WObj:=wPaper;
    MoveL Offs(pOrigin,310.34,207.56,0.00),v40,z0,tPen\WObj:=wPaper;
    MoveL Offs(pOrigin,308.42,204.69,0.00),v40,z0,tPen\WObj:=wPaper;
    MoveL Offs(pOrigin,308.42,205.17,0.00),v40,z0,tPen\WObj:=wPaper;
    MoveL Offs(pOrigin,310.34,207.08,0.00),v40,z0,tPen\WObj:=wPaper;
    MoveL Offs(pOrigin,310.34,207.56,0.00),v40,z0,tPen\WObj:=wPaper;
    MoveL Offs(pOrigin,310.34,206.61,0.00),v40,z0,tPen\WObj:=wPaper;
    MoveL Offs(pOrigin,309.38,205.65,0.00),v40,z0,tPen\WObj:=wPaper;
    MoveL Offs(pOrigin,309.38,206.13,0.00),v40,z0,tPen\WObj:=wPaper;
    MoveL Offs(pOrigin,309.86,206.13,0.00),v40,z0,tPen\WObj:=wPaper;
    MoveL Offs(pOrigin,310.34,206.61,0.00),v40,z0,tPen\WObj:=wPaper;
    MoveL Offs(pOrigin,309.38,205.65,0.00),v40,z0,tPen\WObj:=wPaper;
    MoveL Offs(pOrigin,309.38,206.13,0.00),v40,z0,tPen\WObj:=wPaper;
    MoveL Offs(pOrigin,309.86,206.13,0.00),v40,z0,tPen\WObj:=wPaper;
    MoveL Offs(pOrigin,310.34,206.61,0.00),v40,fine,tPen\WObj:=wPaper;
    MoveL Offs(pOrigin,310.34,206.61,6.00),v60,z5,tPen\WObj:=wPaper;
    MoveL Offs(pOrigin,307.78,204.37,6.00),vTravel,z5,tPen\WObj:=wPaper;
    MoveL Offs(pOrigin,307.78,204.37,0.00),v60,z0,tPen\WObj:=wPaper;
    MoveL Offs(pOrigin,305.55,202.46,0.00),v40,z0,tPen\WObj:=wPaper;
    MoveL Offs(pOrigin,301.40,199.90,0.00),v40,z0,tPen\WObj:=wPaper;
    MoveL Offs(pOrigin,307.78,204.37,0.00),v40,fine,tPen\WObj:=wPaper;
    MoveL Offs(pOrigin,307.78,204.37,6.00),v60,z5,tPen\WObj:=wPaper;
    MoveL Offs(pOrigin,306.51,203.25,6.00),vTravel,z5,tPen\WObj:=wPaper;
    MoveL Offs(pOrigin,306.51,203.25,0.00),v60,z0,tPen\WObj:=wPaper;
    MoveL Offs(pOrigin,305.07,201.82,0.00),v40,z0,tPen\WObj:=wPaper;
    MoveL Offs(pOrigin,305.07,202.30,0.00),v40,z0,tPen\WObj:=wPaper;
    MoveL Offs(pOrigin,305.55,202.30,0.00),v40,z0,tPen\WObj:=wPaper;
    MoveL Offs(pOrigin,306.51,203.25,0.00),v40,z0,tPen\WObj:=wPaper;
    MoveL Offs(pOrigin,305.07,201.82,0.00),v40,z0,tPen\WObj:=wPaper;
    MoveL Offs(pOrigin,305.07,202.30,0.00),v40,z0,tPen\WObj:=wPaper;
    MoveL Offs(pOrigin,305.55,202.30,0.00),v40,z0,tPen\WObj:=wPaper;
    MoveL Offs(pOrigin,306.51,203.25,0.00),v40,fine,tPen\WObj:=wPaper;
    MoveL Offs(pOrigin,306.51,203.25,6.00),v60,z5,tPen\WObj:=wPaper;
    MoveL Offs(pOrigin,304.11,201.34,6.00),vTravel,z5,tPen\WObj:=wPaper;
    MoveL Offs(pOrigin,304.11,201.34,0.00),v60,z0,tPen\WObj:=wPaper;
    MoveL Offs(pOrigin,303.63,200.86,0.00),v40,z0,tPen\WObj:=wPaper;
    MoveL Offs(pOrigin,303.63,201.34,0.00),v40,z0,tPen\WObj:=wPaper;
    MoveL Offs(pOrigin,304.11,201.34,0.00),v40,z0,tPen\WObj:=wPaper;
    MoveL Offs(pOrigin,303.63,200.86,0.00),v40,z0,tPen\WObj:=wPaper;
    MoveL Offs(pOrigin,303.63,201.34,0.00),v40,z0,tPen\WObj:=wPaper;
    MoveL Offs(pOrigin,304.11,201.34,0.00),v40,fine,tPen\WObj:=wPaper;
    MoveL Offs(pOrigin,304.11,201.34,6.00),v60,z5,tPen\WObj:=wPaper;
    MoveL Offs(pOrigin,317.04,193.20,6.00),vTravel,z5,tPen\WObj:=wPaper;
    MoveL Offs(pOrigin,317.04,193.20,0.00),v60,z0,tPen\WObj:=wPaper;
    MoveL Offs(pOrigin,317.04,192.24,0.00),v40,z0,tPen\WObj:=wPaper;
    MoveL Offs(pOrigin,318.00,190.80,0.00),v40,z0,tPen\WObj:=wPaper;
    MoveL Offs(pOrigin,318.00,189.85,0.00),v40,z0,tPen\WObj:=wPaper;
    MoveL Offs(pOrigin,317.04,193.20,0.00),v40,z0,tPen\WObj:=wPaper;
    MoveL Offs(pOrigin,317.04,192.24,0.00),v40,z0,tPen\WObj:=wPaper;
    MoveL Offs(pOrigin,318.00,190.80,0.00),v40,z0,tPen\WObj:=wPaper;
    MoveL Offs(pOrigin,318.00,189.85,0.00),v40,z0,tPen\WObj:=wPaper;
    MoveL Offs(pOrigin,317.04,193.20,0.00),v40,fine,tPen\WObj:=wPaper;
    MoveL Offs(pOrigin,317.04,193.20,6.00),v60,z5,tPen\WObj:=wPaper;
    MoveL Offs(pOrigin,318.48,188.89,6.00),vTravel,z5,tPen\WObj:=wPaper;
    MoveL Offs(pOrigin,318.48,188.89,0.00),v60,z0,tPen\WObj:=wPaper;
    MoveL Offs(pOrigin,319.44,187.93,0.00),v40,z0,tPen\WObj:=wPaper;
    MoveL Offs(pOrigin,319.44,188.41,0.00),v40,z0,tPen\WObj:=wPaper;
    MoveL Offs(pOrigin,318.96,188.41,0.00),v40,z0,tPen\WObj:=wPaper;
    MoveL Offs(pOrigin,318.48,188.89,0.00),v40,z0,tPen\WObj:=wPaper;
    MoveL Offs(pOrigin,319.44,187.93,0.00),v40,z0,tPen\WObj:=wPaper;
    MoveL Offs(pOrigin,319.44,188.41,0.00),v40,z0,tPen\WObj:=wPaper;
    MoveL Offs(pOrigin,318.96,188.41,0.00),v40,z0,tPen\WObj:=wPaper;
    MoveL Offs(pOrigin,318.48,188.89,0.00),v40,fine,tPen\WObj:=wPaper;
    MoveL Offs(pOrigin,318.48,188.89,6.00),v60,z5,tPen\WObj:=wPaper;
    MoveL Offs(pOrigin,319.92,186.97,6.00),vTravel,z5,tPen\WObj:=wPaper;
    MoveL Offs(pOrigin,319.92,186.97,0.00),v60,z0,tPen\WObj:=wPaper;
    MoveL Offs(pOrigin,320.39,186.49,0.00),v40,z0,tPen\WObj:=wPaper;
    MoveL Offs(pOrigin,320.39,186.97,0.00),v40,z0,tPen\WObj:=wPaper;
    MoveL Offs(pOrigin,319.92,186.97,0.00),v40,z0,tPen\WObj:=wPaper;
    MoveL Offs(pOrigin,320.39,186.49,0.00),v40,z0,tPen\WObj:=wPaper;
    MoveL Offs(pOrigin,320.39,186.97,0.00),v40,z0,tPen\WObj:=wPaper;
    MoveL Offs(pOrigin,319.92,186.97,0.00),v40,fine,tPen\WObj:=wPaper;
    MoveL Offs(pOrigin,319.92,186.97,6.00),v60,z5,tPen\WObj:=wPaper;
    MoveL Offs(pOrigin,321.83,184.58,6.00),vTravel,z5,tPen\WObj:=wPaper;
    MoveL Offs(pOrigin,321.83,184.58,0.00),v60,z0,tPen\WObj:=wPaper;
    MoveL Offs(pOrigin,324.23,182.18,0.00),v40,z0,tPen\WObj:=wPaper;
    MoveL Offs(pOrigin,324.23,182.66,0.00),v40,z0,tPen\WObj:=wPaper;
    MoveL Offs(pOrigin,323.75,182.66,0.00),v40,z0,tPen\WObj:=wPaper;
    MoveL Offs(pOrigin,321.83,184.58,0.00),v40,z0,tPen\WObj:=wPaper;
    MoveL Offs(pOrigin,324.23,182.18,0.00),v40,z0,tPen\WObj:=wPaper;
    MoveL Offs(pOrigin,324.23,182.66,0.00),v40,z0,tPen\WObj:=wPaper;
    MoveL Offs(pOrigin,323.75,182.66,0.00),v40,z0,tPen\WObj:=wPaper;
    MoveL Offs(pOrigin,321.83,184.58,0.00),v40,fine,tPen\WObj:=wPaper;
    MoveL Offs(pOrigin,321.83,184.58,6.00),v60,z5,tPen\WObj:=wPaper;
    MoveL Offs(pOrigin,324.70,181.70,6.00),vTravel,z5,tPen\WObj:=wPaper;
    MoveL Offs(pOrigin,324.70,181.70,0.00),v60,z0,tPen\WObj:=wPaper;
    MoveL Offs(pOrigin,325.66,180.75,0.00),v40,z0,tPen\WObj:=wPaper;
    MoveL Offs(pOrigin,325.66,181.23,0.00),v40,z0,tPen\WObj:=wPaper;
  ENDPROC

